LIN {X 0,Y 312.924,Z 444.508,A -85,B 0,C 180,E1 -15752.574,E2 -15752.574} C_VEL
LIN {X 0,Y 312.893,Z 444.512,A -85,B 0,C 180,E1 -15756.448,E2 -15756.448} C_VEL
LIN {X 0,Y 312.698,Z 444.535,A -85,B 0,C 180,E1 -15760.358,E2 -15760.358} C_VEL
LIN {X 0,Y 312.668,Z 444.537,A -85,B 0,C 180,E1 -15764.865,E2 -15764.865} C_VEL
LIN {X 0,Y 312.585,Z 444.545,A -85,B 0,C 180,E1 -15769.212,E2 -15769.212} C_VEL
LIN {X 0,Y 312.525,Z 444.556,A -85,B 0,C 180,E1 -15772.779,E2 -15772.779} C_VEL
LIN {X 0,Y 312.532,Z 444.552,A -85,B 0,C 180,E1 -15775.909,E2 -15775.909} C_VEL
LIN {X 0,Y 312.5,Z 444.556,A -85,B 0,C 180,E1 -15779.654,E2 -15779.654} C_VEL
LIN {X 0,Y 312.519,Z 444.553,A -85,B 0,C 180,E1 -15783.688,E2 -15783.688} C_VEL
LIN {X 0,Y 312.513,Z 444.554,A -85,B 0,C 180,E1 -15787.386,E2 -15787.386} C_VEL
LIN {X 0,Y 312.439,Z 444.567,A -85,B 0,C 180,E1 -15790.717,E2 -15790.717} C_VEL
LIN {X 0,Y 312.45,Z 444.564,A -85,B 0,C 180,E1 -15794.209,E2 -15794.209} C_VEL
LIN {X 0,Y 312.482,Z 444.558,A -85,B 0,C 180,E1 -15797.919,E2 -15797.919} C_VEL
LIN {X 0,Y 312.497,Z 444.558,A -85,B 0,C 180,E1 -15800.971,E2 -15800.971} C_VEL
LIN {X 0,Y 312.531,Z 444.554,A -85,B 0,C 180,E1 -15804.22,E2 -15804.22} C_VEL
LIN {X 0,Y 312.502,Z 444.555,A -85,B 0,C 180,E1 -15807.334,E2 -15807.334} C_VEL
LIN {X 0,Y 312.543,Z 444.55,A -85,B 0,C 180,E1 -15811.279,E2 -15811.279} C_VEL
LIN {X 0,Y 312.584,Z 444.55,A -85,B 0,C 180,E1 -15814.711,E2 -15814.711} C_VEL
LIN {X 0,Y 312.561,Z 444.546,A -85,B 0,C 180,E1 -15817.883,E2 -15817.883} C_VEL
LIN {X 0,Y 311.859,Z 444.638,A -85,B 0,C 180,E1 -15818.959,E2 -15818.959} C_VEL
LIN {X 0,Y 309.003,Z 444.996,A -85,B 0,C 180,E1 -15820.711,E2 -15820.711} C_VEL
LIN {X 0,Y 306.625,Z 445.29,A -85,B 0,C 180,E1 -15822.131,E2 -15822.131} C_VEL
LIN {X 0,Y 305.636,Z 445.412,A -85,B 0,C 180,E1 -15823.231,E2 -15823.231} C_VEL
LIN {X 0,Y 305.57,Z 445.419,A -85,B 0,C 180,E1 -15823.603,E2 -15823.603} C_VEL
LIN {X 0,Y 305.588,Z 445.421,A -85,B 0,C 180,E1 -15826.704,E2 -15826.704} C_VEL
LIN {X 0,Y 305.794,Z 445.392,A -85,B 0,C 180,E1 -15831.21,E2 -15831.21} C_VEL
LIN {X 0,Y 305.84,Z 445.385,A -85,B 0,C 180,E1 -15833.402,E2 -15833.402} C_VEL
LIN {X 0,Y 305.883,Z 445.38,A -85,B 0,C 180,E1 -15837.366,E2 -15837.366} C_VEL
LIN {X 0,Y 306.053,Z 445.359,A -85,B 0,C 180,E1 -15840,E2 -15840} C_VEL
LIN {X 0,Y 305.885,Z 445.385,A -85,B 0,C 180,E1 -15842.634,E2 -15842.634} C_VEL
LIN {X 0,Y 305.852,Z 445.388,A -85,B 0,C 180,E1 -15846.598,E2 -15846.598} C_VEL
LIN {X 0,Y 305.735,Z 445.399,A -85,B 0,C 180,E1 -15849.26,E2 -15849.26} C_VEL
LIN {X 0,Y 305.588,Z 445.417,A -85,B 0,C 180,E1 -15853.296,E2 -15853.296} C_VEL
LIN {X 0,Y 305.593,Z 445.416,A -85,B 0,C 180,E1 -15856.02,E2 -15856.02} C_VEL
LIN {X 0,Y 305.575,Z 445.418,A -85,B 0,C 180,E1 -15859.445,E2 -15859.445} C_VEL
LIN {X 0,Y 305.485,Z 445.431,A -85,B 0,C 180,E1 -15863.04,E2 -15863.04} C_VEL
LIN {X 0,Y 305.553,Z 445.422,A -85,B 0,C 180,E1 -15866.23,E2 -15866.23} C_VEL
LIN {X 0,Y 305.495,Z 445.43,A -85,B 0,C 180,E1 -15869.05,E2 -15869.05} C_VEL
LIN {X 0,Y 305.464,Z 445.432,A -85,B 0,C 180,E1 -15873.517,E2 -15873.517} C_VEL
LIN {X 0,Y 305.474,Z 445.436,A -85,B 0,C 180,E1 -15876.74,E2 -15876.74} C_VEL
LIN {X 0,Y 305.454,Z 445.437,A -85,B 0,C 180,E1 -15880.6,E2 -15880.6} C_VEL
LIN {X 0,Y 305.419,Z 445.441,A -85,B 0,C 180,E1 -15884.493,E2 -15884.493} C_VEL
LIN {X 0,Y 305.442,Z 445.435,A -85,B 0,C 180,E1 -15888.144,E2 -15888.144} C_VEL
LIN {X 0,Y 305.467,Z 445.432,A -85,B 0,C 180,E1 -15891.597,E2 -15891.597} C_VEL
LIN {X 0,Y 305.464,Z 445.437,A -85,B 0,C 180,E1 -15894.888,E2 -15894.888} C_VEL
LIN {X 0,Y 305.504,Z 445.578,A -85,B 0,C 180,E1 -15896.123,E2 -15896.123} C_VEL
LIN {X 0,Y 308.105,Z 458.028,A -85,B 0,C 180,E1 -15899.501,E2 -15899.501} C_VEL
LIN {X 0,Y 310.159,Z 467.904,A -85,B 0,C 180,E1 -15902.094,E2 -15902.094} C_VEL
LIN {X 0,Y 309.465,Z 474.625,A -85,B 0,C 180,E1 -15903.715,E2 -15903.715} C_VEL
LIN {X 0,Y 308.394,Z 483.678,A -85,B 0,C 180,E1 -15905.888,E2 -15905.888} C_VEL
LIN {X 0,Y 313.118,Z 530.091,A -85,B 0,C 180,E1 -15907.613,E2 -15907.613} C_VEL
LIN {X 0,Y 311.173,Z 594.169,A -85,B 0,C 180,E1 -15909.552,E2 -15909.552} C_VEL
LIN {X 0,Y 310.338,Z 607.85,A -85,B 0,C 180,E1 -15910.228,E2 -15910.228} C_VEL
LIN {X 0,Y 309.368,Z 620.327,A -85,B 0,C 180,E1 -15911.112,E2 -15911.112} C_VEL
LIN {X 0,Y 308.299,Z 632.472,A -85,B 0,C 180,E1 -15912.248,E2 -15912.248} C_VEL
LIN {X 0,Y 307.267,Z 643.508,A -85,B 0,C 180,E1 -15913.558,E2 -15913.558} C_VEL
LIN {X 0,Y 306.154,Z 653.974,A -85,B 0,C 180,E1 -15915.115,E2 -15915.115} C_VEL
LIN {X 0,Y 305.413,Z 662.653,A -85,B 0,C 180,E1 -15916.697,E2 -15916.697} C_VEL
LIN {X 0,Y 304.771,Z 670.189,A -85,B 0,C 180,E1 -15918.36,E2 -15918.36} C_VEL
LIN {X 0,Y 304.285,Z 677.561,A -85,B 0,C 180,E1 -15920.361,E2 -15920.361} C_VEL
LIN {X 0,Y 304.075,Z 682.515,A -85,B 0,C 180,E1 -15922.029,E2 -15922.029} C_VEL
LIN {X 0,Y 304.035,Z 687.533,A -85,B 0,C 180,E1 -15924.18,E2 -15924.18} C_VEL
LIN {X 0,Y 303.989,Z 690.733,A -85,B 0,C 180,E1 -15926.023,E2 -15926.023} C_VEL
LIN {X 0,Y 304.153,Z 692.435,A -85,B 0,C 180,E1 -15927.352,E2 -15927.352} C_VEL
LIN {X 0,Y 304.176,Z 693.668,A -85,B 0,C 180,E1 -15928.677,E2 -15928.677} C_VEL
LIN {X 0,Y 304.174,Z 694.458,A -85,B 0,C 180,E1 -15930,E2 -15930} C_VEL
LIN {X 0,Y 304.127,Z 694.76,A -85,B 0,C 180,E1 -15931.325,E2 -15931.325} C_VEL
LIN {X 0,Y 303.936,Z 694.613,A -85,B 0,C 180,E1 -15932.651,E2 -15932.651} C_VEL
LIN {X 0,Y 303.839,Z 694.053,A -85,B 0,C 180,E1 -15933.98,E2 -15933.98} C_VEL
LIN {X 0,Y 303.734,Z 692.62,A -85,B 0,C 180,E1 -15935.75,E2 -15935.75} C_VEL
LIN {X 0,Y 303.932,Z 689.733,A -85,B 0,C 180,E1 -15937.976,E2 -15937.976} C_VEL
LIN {X 0,Y 304.296,Z 686.047,A -85,B 0,C 180,E1 -15939.976,E2 -15939.976} C_VEL
LIN {X 0,Y 304.931,Z 681.285,A -85,B 0,C 180,E1 -15941.972,E2 -15941.972} C_VEL
LIN {X 0,Y 306.073,Z 675.304,A -85,B 0,C 180,E1 -15943.952,E2 -15943.952} C_VEL
LIN {X 0,Y 307.462,Z 667.925,A -85,B 0,C 180,E1 -15945.921,E2 -15945.921} C_VEL
LIN {X 0,Y 309.261,Z 658.8,A -85,B 0,C 180,E1 -15947.866,E2 -15947.866} C_VEL
LIN {X 0,Y 311.407,Z 648.631,A -85,B 0,C 180,E1 -15949.616,E2 -15949.616} C_VEL
LIN {X 0,Y 313.401,Z 638.502,A -85,B 0,C 180,E1 -15951.027,E2 -15951.027} C_VEL
LIN {X 0,Y 315.652,Z 625.934,A -85,B 0,C 180,E1 -15952.414,E2 -15952.414} C_VEL
LIN {X 0,Y 317.702,Z 613.566,A -85,B 0,C 180,E1 -15953.465,E2 -15953.465} C_VEL
LIN {X 0,Y 319.776,Z 598.2,A -85,B 0,C 180,E1 -15954.423,E2 -15954.423} C_VEL
LIN {X 0,Y 320.961,Z 584.573,A -85,B 0,C 180,E1 -15955.017,E2 -15955.017} C_VEL
LIN {X 0,Y 324.197,Z 532.422,A -85,B 0,C 180,E1 -15956.687,E2 -15956.687} C_VEL
LIN {X 0,Y 323.308,Z 519.853,A -85,B 0,C 180,E1 -15957.337,E2 -15957.337} C_VEL
LIN {X 0,Y 321.631,Z 506.064,A -85,B 0,C 180,E1 -15958.198,E2 -15958.198} C_VEL
LIN {X 0,Y 319.141,Z 492.2,A -85,B 0,C 180,E1 -15959.222,E2 -15959.222} C_VEL
LIN {X 0,Y 317.166,Z 483.192,A -85,B 0,C 180,E1 -15959.997,E2 -15959.997} C_VEL
LIN {X 0,Y 315.519,Z 479.419,A -85,B 0,C 180,E1 -15960.479,E2 -15960.479} C_VEL
LIN {X 0,Y 313.437,Z 474.649,A -85,B 0,C 180,E1 -15961.156,E2 -15961.156} C_VEL
LIN {X 0,Y 311.59,Z 466.2,A -85,B 0,C 180,E1 -15964.325,E2 -15964.325} C_VEL
LIN {X 0,Y 310.017,Z 459.968,A -85,B 0,C 180,E1 -15967.003,E2 -15967.003} C_VEL
LIN {X 0,Y 308.169,Z 453.871,A -85,B 0,C 180,E1 -15970.092,E2 -15970.092} C_VEL
LIN {X 0,Y 306.421,Z 448.344,A -85,B 0,C 180,E1 -15973.479,E2 -15973.479} C_VEL
LIN {X 0,Y 305.432,Z 445.437,A -85,B 0,C 180,E1 -15975.77,E2 -15975.77} C_VEL
LIN {X 0,Y 305.458,Z 445.433,A -85,B 0,C 180,E1 -15979.4,E2 -15979.4} C_VEL
LIN {X 0,Y 305.5,Z 445.427,A -85,B 0,C 180,E1 -15983.264,E2 -15983.264} C_VEL
LIN {X 0,Y 305.468,Z 445.435,A -85,B 0,C 180,E1 -15986.483,E2 -15986.483} C_VEL
LIN {X 0,Y 305.434,Z 445.435,A -85,B 0,C 180,E1 -15989.588,E2 -15989.588} C_VEL
LIN {X 0,Y 305.455,Z 445.437,A -85,B 0,C 180,E1 -15992.602,E2 -15992.602} C_VEL
LIN {X 0,Y 305.444,Z 445.436,A -85,B 0,C 180,E1 -15995.533,E2 -15995.533} C_VEL
LIN {X 0,Y 305.469,Z 445.479,A -85,B 0,C 180,E1 -15999.46,E2 -15999.46} C_VEL
LIN {X 0,Y 306.697,Z 449.416,A -85,B 0,C 180,E1 -16002.556,E2 -16002.556} C_VEL
LIN {X 0,Y 309.371,Z 453.214,A -85,B 0,C 180,E1 -16003.392,E2 -16003.392} C_VEL
LIN {X 0,Y 313.552,Z 459.105,A -85,B 0,C 180,E1 -16004.611,E2 -16004.611} C_VEL
LIN {X 0,Y 318.191,Z 466.055,A -85,B 0,C 180,E1 -16005.849,E2 -16005.849} C_VEL
LIN {X 0,Y 323.55,Z 475.549,A -85,B 0,C 180,E1 -16007.23,E2 -16007.23} C_VEL
LIN {X 0,Y 326.691,Z 482.075,A -85,B 0,C 180,E1 -16008.019,E2 -16008.019} C_VEL
LIN {X 0,Y 322.133,Z 551.699,A -85,B 0,C 180,E1 -16010.315,E2 -16010.315} C_VEL
LIN {X 0,Y 321.025,Z 566.069,A -85,B 0,C 180,E1 -16011.077,E2 -16011.077} C_VEL
LIN {X 0,Y 319.611,Z 579.113,A -85,B 0,C 180,E1 -16012.061,E2 -16012.061} C_VEL
LIN {X 0,Y 317.777,Z 591.737,A -85,B 0,C 180,E1 -16013.3,E2 -16013.3} C_VEL
LIN {X 0,Y 315.868,Z 603.067,A -85,B 0,C 180,E1 -16014.734,E2 -16014.734} C_VEL
LIN {X 0,Y 314.132,Z 612.119,A -85,B 0,C 180,E1 -16016.151,E2 -16016.151} C_VEL
LIN {X 0,Y 312.36,Z 620.449,A -85,B 0,C 180,E1 -16017.743,E2 -16017.743} C_VEL
LIN {X 0,Y 310.485,Z 628.539,A -85,B 0,C 180,E1 -16019.676,E2 -16019.676} C_VEL
LIN {X 0,Y 309.133,Z 634.088,A -85,B 0,C 180,E1 -16021.303,E2 -16021.303} C_VEL
LIN {X 0,Y 307.742,Z 639.484,A -85,B 0,C 180,E1 -16023.273,E2 -16023.273} C_VEL
LIN {X 0,Y 306.615,Z 643.66,A -85,B 0,C 180,E1 -16025.26,E2 -16025.26} C_VEL
LIN {X 0,Y 305.971,Z 645.843,A -85,B 0,C 180,E1 -16026.595,E2 -16026.595} C_VEL
LIN {X 0,Y 305.338,Z 647.82,A -85,B 0,C 180,E1 -16028.212,E2 -16028.212} C_VEL
LIN {X 0,Y 304.626,Z 649.586,A -85,B 0,C 180,E1 -16030.636,E2 -16030.636} C_VEL
LIN {X 0,Y 304.334,Z 649.967,A -85,B 0,C 180,E1 -16031.996,E2 -16031.996} C_VEL
LIN {X 0,Y 304.122,Z 649.714,A -85,B 0,C 180,E1 -16033.929,E2 -16033.929} C_VEL
LIN {X 0,Y 303.964,Z 648.349,A -85,B 0,C 180,E1 -16036.108,E2 -16036.108} C_VEL
LIN {X 0,Y 304.078,Z 645.291,A -85,B 0,C 180,E1 -16038.626,E2 -16038.626} C_VEL
LIN {X 0,Y 304.375,Z 640.985,A -85,B 0,C 180,E1 -16040.971,E2 -16040.971} C_VEL
LIN {X 0,Y 304.755,Z 635.706,A -85,B 0,C 180,E1 -16043.081,E2 -16043.081} C_VEL
LIN {X 0,Y 305.379,Z 628.903,A -85,B 0,C 180,E1 -16045.199,E2 -16045.199} C_VEL
LIN {X 0,Y 306.085,Z 621.556,A -85,B 0,C 180,E1 -16047.039,E2 -16047.039} C_VEL
LIN {X 0,Y 306.861,Z 613.232,A -85,B 0,C 180,E1 -16048.748,E2 -16048.748} C_VEL
LIN {X 0,Y 307.785,Z 603.69,A -85,B 0,C 180,E1 -16050.345,E2 -16050.345} C_VEL
LIN {X 0,Y 308.699,Z 593.276,A -85,B 0,C 180,E1 -16051.768,E2 -16051.768} C_VEL
LIN {X 0,Y 309.632,Z 582.052,A -85,B 0,C 180,E1 -16053.008,E2 -16053.008} C_VEL
LIN {X 0,Y 310.479,Z 569.679,A -85,B 0,C 180,E1 -16054.072,E2 -16054.072} C_VEL
LIN {X 0,Y 311.252,Z 555.875,A -85,B 0,C 180,E1 -16054.957,E2 -16054.957} C_VEL
LIN {X 0,Y 311.664,Z 543.598,A -85,B 0,C 180,E1 -16055.497,E2 -16055.497} C_VEL
LIN {X 0,Y 313.908,Z 469.49,A -85,B 0,C 180,E1 -16057.692,E2 -16057.692} C_VEL
LIN {X 0,Y 305.459,Z 445.434,A -85,B 0,C 180,E1 -16058.935,E2 -16058.935} C_VEL
LIN {X 0,Y 305.438,Z 445.439,A -85,B 0,C 180,E1 -16062.581,E2 -16062.581} C_VEL
LIN {X 0,Y 305.427,Z 445.442,A -85,B 0,C 180,E1 -16066.344,E2 -16066.344} C_VEL
LIN {X 0,Y 305.412,Z 445.44,A -85,B 0,C 180,E1 -16069.884,E2 -16069.884} C_VEL
LIN {X 0,Y 305.464,Z 445.432,A -85,B 0,C 180,E1 -16073.636,E2 -16073.636} C_VEL
LIN {X 0,Y 305.467,Z 445.437,A -85,B 0,C 180,E1 -16076.483,E2 -16076.483} C_VEL
LIN {X 0,Y 305.432,Z 445.436,A -85,B 0,C 180,E1 -16079.587,E2 -16079.587} C_VEL
LIN {X 0,Y 305.459,Z 445.436,A -85,B 0,C 180,E1 -16082.602,E2 -16082.602} C_VEL
LIN {X 0,Y 305.487,Z 445.429,A -85,B 0,C 180,E1 -16085.536,E2 -16085.536} C_VEL
LIN {X 0,Y 305.519,Z 445.426,A -85,B 0,C 180,E1 -16089.814,E2 -16089.814} C_VEL
LIN {X 0,Y 305.576,Z 445.422,A -85,B 0,C 180,E1 -16092.603,E2 -16092.603} C_VEL
LIN {X 0,Y 305.651,Z 445.409,A -85,B 0,C 180,E1 -16095.349,E2 -16095.349} C_VEL
LIN {X 0,Y 305.626,Z 445.411,A -85,B 0,C 180,E1 -16099.399,E2 -16099.399} C_VEL
LIN {X 0,Y 305.748,Z 445.398,A -85,B 0,C 180,E1 -16102.072,E2 -16102.072} C_VEL
LIN {X 0,Y 305.668,Z 445.41,A -85,B 0,C 180,E1 -16104.723,E2 -16104.723} C_VEL
LIN {X 0,Y 305.952,Z 445.374,A -85,B 0,C 180,E1 -16108.683,E2 -16108.683} C_VEL
LIN {X 0,Y 305.953,Z 445.371,A -85,B 0,C 180,E1 -16111.316,E2 -16111.316} C_VEL
LIN {X 0,Y 305.833,Z 445.39,A -85,B 0,C 180,E1 -16116.597,E2 -16116.597} C_VEL
LIN {X 0,Y 305.698,Z 445.403,A -85,B 0,C 180,E1 -16119.26,E2 -16119.26} C_VEL
LIN {X 0,Y 305.588,Z 445.417,A -85,B 0,C 180,E1 -16123.296,E2 -16123.296} C_VEL
LIN {X 0,Y 305.552,Z 445.422,A -85,B 0,C 180,E1 -16126.022,E2 -16126.022} C_VEL
LIN {X 0,Y 305.542,Z 445.422,A -85,B 0,C 180,E1 -16129.426,E2 -16129.426} C_VEL
LIN {X 0,Y 305.486,Z 445.43,A -85,B 0,C 180,E1 -16133.039,E2 -16133.039} C_VEL
LIN {X 0,Y 305.472,Z 445.433,A -85,B 0,C 180,E1 -16136.198,E2 -16136.198} C_VEL
LIN {X 0,Y 305.458,Z 445.434,A -85,B 0,C 180,E1 -16139.037,E2 -16139.037} C_VEL
LIN {X 0,Y 305.436,Z 445.436,A -85,B 0,C 180,E1 -16141.953,E2 -16141.953} C_VEL
LIN {X 0,Y 305.461,Z 445.433,A -85,B 0,C 180,E1 -16145.113,E2 -16145.113} C_VEL
LIN {X 0,Y 305.433,Z 445.441,A -85,B 0,C 180,E1 -16148.525,E2 -16148.525} C_VEL
LIN {X 0,Y 305.435,Z 445.441,A -85,B 0,C 180,E1 -16152.582,E2 -16152.582} C_VEL
LIN {X 0,Y 305.424,Z 445.44,A -85,B 0,C 180,E1 -16156.345,E2 -16156.345} C_VEL
LIN {X 0,Y 305.457,Z 445.433,A -85,B 0,C 180,E1 -16159.892,E2 -16159.892} C_VEL
LIN {X 0,Y 305.479,Z 445.43,A -85,B 0,C 180,E1 -16163.632,E2 -16163.632} C_VEL
LIN {X 0,Y 305.464,Z 445.437,A -85,B 0,C 180,E1 -16166.483,E2 -16166.483} C_VEL
LIN {X 0,Y 305.457,Z 445.432,A -85,B 0,C 180,E1 -16169.59,E2 -16169.59} C_VEL
LIN {X 0,Y 305.514,Z 445.431,A -85,B 0,C 180,E1 -16172.608,E2 -16172.608} C_VEL
LIN {X 0,Y 305.507,Z 445.427,A -85,B 0,C 180,E1 -16175.539,E2 -16175.539} C_VEL
LIN {X 0,Y 305.519,Z 445.425,A -85,B 0,C 180,E1 -16179.815,E2 -16179.815} C_VEL
LIN {X 0,Y 305.574,Z 445.424,A -85,B 0,C 180,E1 -16182.603,E2 -16182.603} C_VEL
LIN {X 0,Y 305.57,Z 445.419,A -85,B 0,C 180,E1 -16183.603,E2 -16183.603} C_VEL
LIN {X 0,Y 304.941,Z 445.502,A -85,B 0,C 180,E1 -16184.703,E2 -16184.703} C_VEL
LIN {X 0,Y 302.103,Z 445.855,A -85,B 0,C 180,E1 -16186.493,E2 -16186.493} C_VEL
LIN {X 0,Y 299.687,Z 446.154,A -85,B 0,C 180,E1 -16187.946,E2 -16187.946} C_VEL
LIN {X 0,Y 298.669,Z 446.281,A -85,B 0,C 180,E1 -16189.071,E2 -16189.071} C_VEL
LIN {X 0,Y 298.597,Z 446.287,A -85,B 0,C 180,E1 -16189.452,E2 -16189.452} C_VEL
LIN {X 0,Y 298.751,Z 446.269,A -85,B 0,C 180,E1 -16191.886,E2 -16191.886} C_VEL
LIN {X 0,Y 298.652,Z 446.286,A -85,B 0,C 180,E1 -16194.599,E2 -16194.599} C_VEL
LIN {X 0,Y 298.921,Z 446.252,A -85,B 0,C 180,E1 -16198.653,E2 -16198.653} C_VEL
LIN {X 0,Y 298.922,Z 446.247,A -85,B 0,C 180,E1 -16201.347,E2 -16201.347} C_VEL
LIN {X 0,Y 298.797,Z 446.267,A -85,B 0,C 180,E1 -16206.754,E2 -16206.754} C_VEL
LIN {X 0,Y 298.68,Z 446.277,A -85,B 0,C 180,E1 -16209.481,E2 -16209.481} C_VEL
LIN {X 0,Y 298.552,Z 446.292,A -85,B 0,C 180,E1 -16213.616,E2 -16213.616} C_VEL
LIN {X 0,Y 298.548,Z 446.296,A -85,B 0,C 180,E1 -16216.409,E2 -16216.409} C_VEL
LIN {X 0,Y 298.509,Z 446.298,A -85,B 0,C 180,E1 -16219.654,E2 -16219.654} C_VEL
LIN {X 0,Y 298.428,Z 446.308,A -85,B 0,C 180,E1 -16223.6,E2 -16223.6} C_VEL
LIN {X 0,Y 298.491,Z 446.305,A -85,B 0,C 180,E1 -16226.574,E2 -16226.574} C_VEL
LIN {X 0,Y 298.42,Z 446.309,A -85,B 0,C 180,E1 -16229.641,E2 -16229.641} C_VEL
LIN {X 0,Y 298.395,Z 446.317,A -85,B 0,C 180,E1 -16232.8,E2 -16232.8} C_VEL
LIN {X 0,Y 298.446,Z 446.311,A -85,B 0,C 180,E1 -16236.808,E2 -16236.808} C_VEL
LIN {X 0,Y 298.387,Z 446.316,A -85,B 0,C 180,E1 -16241.088,E2 -16241.088} C_VEL
LIN {X 0,Y 298.388,Z 446.316,A -85,B 0,C 180,E1 -16245.042,E2 -16245.042} C_VEL
LIN {X 0,Y 298.388,Z 446.317,A -85,B 0,C 180,E1 -16248.912,E2 -16248.912} C_VEL
LIN {X 0,Y 298.444,Z 446.309,A -85,B 0,C 180,E1 -16253.193,E2 -16253.193} C_VEL
LIN {X 0,Y 298.443,Z 446.464,A -85,B 0,C 180,E1 -16255.841,E2 -16255.841} C_VEL
LIN {X 0,Y 300.859,Z 458.098,A -85,B 0,C 180,E1 -16259.075,E2 -16259.075} C_VEL
LIN {X 0,Y 303.146,Z 468.868,A -85,B 0,C 180,E1 -16261.976,E2 -16261.976} C_VEL
LIN {X 0,Y 301.624,Z 481.991,A -85,B 0,C 180,E1 -16265.203,E2 -16265.203} C_VEL
LIN {X 0,Y 301.479,Z 483.267,A -85,B 0,C 180,E1 -16265.516,E2 -16265.516} C_VEL
LIN {X 0,Y 306.2,Z 531.288,A -85,B 0,C 180,E1 -16267.332,E2 -16267.332} C_VEL
LIN {X 0,Y 304.233,Z 593.859,A -85,B 0,C 180,E1 -16269.285,E2 -16269.285} C_VEL
LIN {X 0,Y 303.443,Z 606.759,A -85,B 0,C 180,E1 -16269.936,E2 -16269.936} C_VEL
LIN {X 0,Y 302.437,Z 619.395,A -85,B 0,C 180,E1 -16270.839,E2 -16270.839} C_VEL
LIN {X 0,Y 301.337,Z 631.609,A -85,B 0,C 180,E1 -16272,E2 -16272} C_VEL
LIN {X 0,Y 300.273,Z 642.717,A -85,B 0,C 180,E1 -16273.339,E2 -16273.339} C_VEL
LIN {X 0,Y 299.084,Z 653.754,A -85,B 0,C 180,E1 -16275.02,E2 -16275.02} C_VEL
LIN {X 0,Y 298.295,Z 662.772,A -85,B 0,C 180,E1 -16276.72,E2 -16276.72} C_VEL
LIN {X 0,Y 297.667,Z 670.193,A -85,B 0,C 180,E1 -16278.423,E2 -16278.423} C_VEL
LIN {X 0,Y 297.193,Z 677.42,A -85,B 0,C 180,E1 -16280.472,E2 -16280.472} C_VEL
LIN {X 0,Y 297.001,Z 683.144,A -85,B 0,C 180,E1 -16282.522,E2 -16282.522} C_VEL
LIN {X 0,Y 297.002,Z 687.565,A -85,B 0,C 180,E1 -16284.569,E2 -16284.569} C_VEL
LIN {X 0,Y 296.928,Z 689.844,A -85,B 0,C 180,E1 -16285.929,E2 -16285.929} C_VEL
LIN {X 0,Y 297.077,Z 691.633,A -85,B 0,C 180,E1 -16287.289,E2 -16287.289} C_VEL
LIN {X 0,Y 297.118,Z 692.919,A -85,B 0,C 180,E1 -16288.645,E2 -16288.645} C_VEL
LIN {X 0,Y 297.115,Z 693.762,A -85,B 0,C 180,E1 -16290,E2 -16290} C_VEL
LIN {X 0,Y 297.064,Z 694.158,A -85,B 0,C 180,E1 -16291.356,E2 -16291.356} C_VEL
LIN {X 0,Y 296.845,Z 694.062,A -85,B 0,C 180,E1 -16292.715,E2 -16292.715} C_VEL
LIN {X 0,Y 296.762,Z 693.548,A -85,B 0,C 180,E1 -16294.075,E2 -16294.075} C_VEL
LIN {X 0,Y 296.667,Z 692.351,A -85,B 0,C 180,E1 -16295.745,E2 -16295.745} C_VEL
LIN {X 0,Y 296.863,Z 689.43,A -85,B 0,C 180,E1 -16298.167,E2 -16298.167} C_VEL
LIN {X 0,Y 297.264,Z 685.872,A -85,B 0,C 180,E1 -16300.214,E2 -16300.214} C_VEL
LIN {X 0,Y 297.959,Z 681.219,A -85,B 0,C 180,E1 -16302.257,E2 -16302.257} C_VEL
LIN {X 0,Y 299.404,Z 674.255,A -85,B 0,C 180,E1 -16304.616,E2 -16304.616} C_VEL
LIN {X 0,Y 300.83,Z 667.312,A -85,B 0,C 180,E1 -16306.505,E2 -16306.505} C_VEL
LIN {X 0,Y 302.537,Z 659.349,A -85,B 0,C 180,E1 -16308.277,E2 -16308.277} C_VEL
LIN {X 0,Y 304.784,Z 649.381,A -85,B 0,C 180,E1 -16310.06,E2 -16310.06} C_VEL
LIN {X 0,Y 307.109,Z 638.319,A -85,B 0,C 180,E1 -16311.655,E2 -16311.655} C_VEL
LIN {X 0,Y 309.476,Z 625.993,A -85,B 0,C 180,E1 -16313.063,E2 -16313.063} C_VEL
LIN {X 0,Y 311.639,Z 613.954,A -85,B 0,C 180,E1 -16314.127,E2 -16314.127} C_VEL
LIN {X 0,Y 313.627,Z 600.459,A -85,B 0,C 180,E1 -16315.023,E2 -16315.023} C_VEL
LIN {X 0,Y 315.051,Z 586.508,A -85,B 0,C 180,E1 -16315.697,E2 -16315.697} C_VEL
LIN {X 0,Y 318.587,Z 534.067,A -85,B 0,C 180,E1 -16317.428,E2 -16317.428} C_VEL
LIN {X 0,Y 317.987,Z 522.485,A -85,B 0,C 180,E1 -16318.035,E2 -16318.035} C_VEL
LIN {X 0,Y 316.341,Z 508.34,A -85,B 0,C 180,E1 -16318.939,E2 -16318.939} C_VEL
LIN {X 0,Y 314.019,Z 494.453,A -85,B 0,C 180,E1 -16320.014,E2 -16320.014} C_VEL
LIN {X 0,Y 312.378,Z 486.751,A -85,B 0,C 180,E1 -16320.702,E2 -16320.702} C_VEL
LIN {X 0,Y 308.856,Z 479.015,A -85,B 0,C 180,E1 -16321.805,E2 -16321.805} C_VEL
LIN {X 0,Y 306.34,Z 474.117,A -85,B 0,C 180,E1 -16322.609,E2 -16322.609} C_VEL
LIN {X 0,Y 306.161,Z 473.602,A -85,B 0,C 180,E1 -16322.695,E2 -16322.695} C_VEL
LIN {X 0,Y 304.804,Z 467.402,A -85,B 0,C 180,E1 -16325.201,E2 -16325.201} C_VEL
LIN {X 0,Y 303.165,Z 461.414,A -85,B 0,C 180,E1 -16327.983,E2 -16327.983} C_VEL
LIN {X 0,Y 301.658,Z 456.346,A -85,B 0,C 180,E1 -16330.719,E2 -16330.719} C_VEL
LIN {X 0,Y 300.327,Z 452.028,A -85,B 0,C 180,E1 -16333.495,E2 -16333.495} C_VEL
LIN {X 0,Y 298.785,Z 447.863,A -85,B 0,C 180,E1 -16336.989,E2 -16336.989} C_VEL
LIN {X 0,Y 298.416,Z 446.312,A -85,B 0,C 180,E1 -16338.743,E2 -16338.743} C_VEL
LIN {X 0,Y 298.435,Z 446.312,A -85,B 0,C 180,E1 -16342.245,E2 -16342.245} C_VEL
LIN {X 0,Y 298.412,Z 446.309,A -85,B 0,C 180,E1 -16345.581,E2 -16345.581} C_VEL
LIN {X 0,Y 298.381,Z 446.317,A -85,B 0,C 180,E1 -16348.789,E2 -16348.789} C_VEL
LIN {X 0,Y 298.414,Z 446.31,A -85,B 0,C 180,E1 -16351.899,E2 -16351.899} C_VEL
LIN {X 0,Y 298.417,Z 446.315,A -85,B 0,C 180,E1 -16354.918,E2 -16354.918} C_VEL
LIN {X 0,Y 298.41,Z 446.414,A -85,B 0,C 180,E1 -16356.711,E2 -16356.711} C_VEL
LIN {X 0,Y 299.391,Z 449.481,A -85,B 0,C 180,E1 -16359.881,E2 -16359.881} C_VEL
LIN {X 0,Y 299.822,Z 450.694,A -85,B 0,C 180,E1 -16360.867,E2 -16360.867} C_VEL
LIN {X 0,Y 302.605,Z 454.462,A -85,B 0,C 180,E1 -16361.844,E2 -16361.844} C_VEL
LIN {X 0,Y 304.477,Z 457.05,A -85,B 0,C 180,E1 -16362.474,E2 -16362.474} C_VEL
LIN {X 0,Y 309.201,Z 463.406,A -85,B 0,C 180,E1 -16363.922,E2 -16363.922} C_VEL
LIN {X 0,Y 315.613,Z 473.663,A -85,B 0,C 180,E1 -16365.754,E2 -16365.754} C_VEL
LIN {X 0,Y 321.198,Z 484.416,A -85,B 0,C 180,E1 -16367.252,E2 -16367.252} C_VEL
LIN {X 0,Y 316.456,Z 552.323,A -85,B 0,C 180,E1 -16369.564,E2 -16369.564} C_VEL
LIN {X 0,Y 315.338,Z 565.985,A -85,B 0,C 180,E1 -16370.297,E2 -16370.297} C_VEL
LIN {X 0,Y 313.952,Z 578.602,A -85,B 0,C 180,E1 -16371.24,E2 -16371.24} C_VEL
LIN {X 0,Y 312.101,Z 590.826,A -85,B 0,C 180,E1 -16372.426,E2 -16372.426} C_VEL
LIN {X 0,Y 310.094,Z 602.033,A -85,B 0,C 180,E1 -16373.82,E2 -16373.82} C_VEL
LIN {X 0,Y 308.016,Z 612.21,A -85,B 0,C 180,E1 -16375.419,E2 -16375.419} C_VEL
LIN {X 0,Y 306.068,Z 620.669,A -85,B 0,C 180,E1 -16377.038,E2 -16377.038} C_VEL
LIN {X 0,Y 304.116,Z 628.855,A -85,B 0,C 180,E1 -16379.007,E2 -16379.007} C_VEL
LIN {X 0,Y 302.268,Z 635.854,A -85,B 0,C 180,E1 -16381.145,E2 -16381.145} C_VEL
LIN {X 0,Y 300.687,Z 641.419,A -85,B 0,C 180,E1 -16383.35,E2 -16383.35} C_VEL
LIN {X 0,Y 299.513,Z 645.28,A -85,B 0,C 180,E1 -16385.386,E2 -16385.386} C_VEL
LIN {X 0,Y 298.865,Z 647.225,A -85,B 0,C 180,E1 -16386.752,E2 -16386.752} C_VEL
LIN {X 0,Y 298.263,Z 648.853,A -85,B 0,C 180,E1 -16388.246,E2 -16388.246} C_VEL
LIN {X 0,Y 297.863,Z 649.81,A -85,B 0,C 180,E1 -16389.507,E2 -16389.507} C_VEL
LIN {X 0,Y 297.487,Z 650.404,A -85,B 0,C 180,E1 -16390.894,E2 -16390.894} C_VEL
LIN {X 0,Y 297.23,Z 650.572,A -85,B 0,C 180,E1 -16392.287,E2 -16392.287} C_VEL
LIN {X 0,Y 297.043,Z 650.148,A -85,B 0,C 180,E1 -16394.054,E2 -16394.054} C_VEL
LIN {X 0,Y 296.871,Z 648.371,A -85,B 0,C 180,E1 -16396.504,E2 -16396.504} C_VEL
LIN {X 0,Y 296.999,Z 645.396,A -85,B 0,C 180,E1 -16398.818,E2 -16398.818} C_VEL
LIN {X 0,Y 297.249,Z 641.809,A -85,B 0,C 180,E1 -16400.772,E2 -16400.772} C_VEL
LIN {X 0,Y 297.668,Z 636.551,A -85,B 0,C 180,E1 -16402.956,E2 -16402.956} C_VEL
LIN {X 0,Y 298.234,Z 629.886,A -85,B 0,C 180,E1 -16405.099,E2 -16405.099} C_VEL
LIN {X 0,Y 299.09,Z 621.376,A -85,B 0,C 180,E1 -16407.271,E2 -16407.271} C_VEL
LIN {X 0,Y 299.928,Z 612.441,A -85,B 0,C 180,E1 -16409.092,E2 -16409.092} C_VEL
LIN {X 0,Y 300.872,Z 603.012,A -85,B 0,C 180,E1 -16410.666,E2 -16410.666} C_VEL
LIN {X 0,Y 301.864,Z 591.901,A -85,B 0,C 180,E1 -16412.18,E2 -16412.18} C_VEL
LIN {X 0,Y 302.795,Z 579.942,A -85,B 0,C 180,E1 -16413.466,E2 -16413.466} C_VEL
LIN {X 0,Y 303.697,Z 567.093,A -85,B 0,C 180,E1 -16414.539,E2 -16414.539} C_VEL
LIN {X 0,Y 304.395,Z 553.024,A -85,B 0,C 180,E1 -16415.385,E2 -16415.385} C_VEL
LIN {X 0,Y 304.885,Z 539.253,A -85,B 0,C 180,E1 -16415.931,E2 -16415.931} C_VEL
LIN {X 0,Y 307.052,Z 470.895,A -85,B 0,C 180,E1 -16418.007,E2 -16418.007} C_VEL
LIN {X 0,Y 298.408,Z 446.311,A -85,B 0,C 180,E1 -16419.3,E2 -16419.3} C_VEL
LIN {X 0,Y 298.373,Z 446.316,A -85,B 0,C 180,E1 -16423.097,E2 -16423.097} C_VEL
LIN {X 0,Y 298.405,Z 446.312,A -85,B 0,C 180,E1 -16426.92,E2 -16426.92} C_VEL
LIN {X 0,Y 298.358,Z 446.318,A -85,B 0,C 180,E1 -16431.017,E2 -16431.017} C_VEL
LIN {X 0,Y 298.407,Z 446.312,A -85,B 0,C 180,E1 -16433.928,E2 -16433.928} C_VEL
LIN {X 0,Y 298.395,Z 446.313,A -85,B 0,C 180,E1 -16437.199,E2 -16437.199} C_VEL
LIN {X 0,Y 298.404,Z 446.315,A -85,B 0,C 180,E1 -16440.625,E2 -16440.625} C_VEL
LIN {X 0,Y 298.447,Z 446.307,A -85,B 0,C 180,E1 -16444.92,E2 -16444.92} C_VEL
LIN {X 0,Y 298.45,Z 446.306,A -85,B 0,C 180,E1 -16449.315,E2 -16449.315} C_VEL
LIN {X 0,Y 298.54,Z 446.297,A -85,B 0,C 180,E1 -16452.179,E2 -16452.179} C_VEL
LIN {X 0,Y 298.595,Z 446.289,A -85,B 0,C 180,E1 -16454.994,E2 -16454.994} C_VEL
LIN {X 0,Y 298.585,Z 446.289,A -85,B 0,C 180,E1 -16459.146,E2 -16459.146} C_VEL
LIN {X 0,Y 298.699,Z 446.275,A -85,B 0,C 180,E1 -16461.884,E2 -16461.884} C_VEL
LIN {X 0,Y 298.637,Z 446.287,A -85,B 0,C 180,E1 -16464.598,E2 -16464.598} C_VEL
LIN {X 0,Y 298.919,Z 446.25,A -85,B 0,C 180,E1 -16468.652,E2 -16468.652} C_VEL
LIN {X 0,Y 298.919,Z 446.247,A -85,B 0,C 180,E1 -16471.347,E2 -16471.347} C_VEL
LIN {X 0,Y 298.777,Z 446.267,A -85,B 0,C 180,E1 -16476.754,E2 -16476.754} C_VEL
LIN {X 0,Y 298.631,Z 446.283,A -85,B 0,C 180,E1 -16479.482,E2 -16479.482} C_VEL
LIN {X 0,Y 298.546,Z 446.294,A -85,B 0,C 180,E1 -16483.615,E2 -16483.615} C_VEL
LIN {X 0,Y 298.487,Z 446.305,A -85,B 0,C 180,E1 -16486.412,E2 -16486.412} C_VEL
LIN {X 0,Y 298.483,Z 446.302,A -85,B 0,C 180,E1 -16489.639,E2 -16489.639} C_VEL
LIN {X 0,Y 298.423,Z 446.309,A -85,B 0,C 180,E1 -16493.6,E2 -16493.6} C_VEL
LIN {X 0,Y 298.412,Z 446.315,A -85,B 0,C 180,E1 -16496.581,E2 -16496.581} C_VEL
LIN {X 0,Y 298.397,Z 446.312,A -85,B 0,C 180,E1 -16499.643,E2 -16499.643} C_VEL
LIN {X 0,Y 298.392,Z 446.315,A -85,B 0,C 180,E1 -16502.8,E2 -16502.8} C_VEL
LIN {X 0,Y 298.441,Z 446.31,A -85,B 0,C 180,E1 -16506.806,E2 -16506.806} C_VEL
LIN {X 0,Y 298.347,Z 446.319,A -85,B 0,C 180,E1 -16511.079,E2 -16511.079} C_VEL
LIN {X 0,Y 298.398,Z 446.313,A -85,B 0,C 180,E1 -16513.103,E2 -16513.103} C_VEL
LIN {X 0,Y 298.402,Z 446.314,A -85,B 0,C 180,E1 -16516.92,E2 -16516.92} C_VEL
LIN {X 0,Y 298.397,Z 446.313,A -85,B 0,C 180,E1 -16521.007,E2 -16521.007} C_VEL
LIN {X 0,Y 298.417,Z 446.31,A -85,B 0,C 180,E1 -16523.93,E2 -16523.93} C_VEL
LIN {X 0,Y 298.392,Z 446.314,A -85,B 0,C 180,E1 -16527.984,E2 -16527.984} C_VEL
LIN {X 0,Y 298.456,Z 446.305,A -85,B 0,C 180,E1 -16531.904,E2 -16531.904} C_VEL
LIN {X 0,Y 298.482,Z 446.304,A -85,B 0,C 180,E1 -16534.924,E2 -16534.924} C_VEL
LIN {X 0,Y 298.45,Z 446.306,A -85,B 0,C 180,E1 -16539.315,E2 -16539.315} C_VEL
LIN {X 0,Y 298.537,Z 446.297,A -85,B 0,C 180,E1 -16542.179,E2 -16542.179} C_VEL
LIN {X 0,Y 298.593,Z 446.29,A -85,B 0,C 180,E1 -16544.995,E2 -16544.995} C_VEL
LIN {X 0,Y 298.597,Z 446.287,A -85,B 0,C 180,E1 -16549.452,E2 -16549.452} C_VEL
LIN {X 0,Y 297.962,Z 446.371,A -85,B 0,C 180,E1 -16550.58,E2 -16550.58} C_VEL
LIN {X 0,Y 295.129,Z 446.723,A -85,B 0,C 180,E1 -16552.416,E2 -16552.416} C_VEL
LIN {X 0,Y 292.699,Z 447.023,A -85,B 0,C 180,E1 -16553.906,E2 -16553.906} C_VEL
LIN {X 0,Y 291.644,Z 447.155,A -85,B 0,C 180,E1 -16555.06,E2 -16555.06} C_VEL
LIN {X 0,Y 291.552,Z 447.164,A -85,B 0,C 180,E1 -16555.452,E2 -16555.452} C_VEL
LIN {X 0,Y 291.888,Z 447.128,A -85,B 0,C 180,E1 -16558.62,E2 -16558.62} C_VEL
LIN {X 0,Y 291.888,Z 447.124,A -85,B 0,C 180,E1 -16561.38,E2 -16561.38} C_VEL
LIN {X 0,Y 291.746,Z 447.144,A -85,B 0,C 180,E1 -16566.918,E2 -16566.918} C_VEL
LIN {X 0,Y 291.629,Z 447.156,A -85,B 0,C 180,E1 -16569.712,E2 -16569.712} C_VEL
LIN {X 0,Y 291.521,Z 447.168,A -85,B 0,C 180,E1 -16573.95,E2 -16573.95} C_VEL
LIN {X 0,Y 291.487,Z 447.177,A -85,B 0,C 180,E1 -16576.818,E2 -16576.818} C_VEL
LIN {X 0,Y 291.45,Z 447.178,A -85,B 0,C 180,E1 -16579.875,E2 -16579.875} C_VEL
LIN {X 0,Y 291.382,Z 447.187,A -85,B 0,C 180,E1 -16584.207,E2 -16584.207} C_VEL
LIN {X 0,Y 291.425,Z 447.182,A -85,B 0,C 180,E1 -16587.271,E2 -16587.271} C_VEL
LIN {X 0,Y 291.337,Z 447.194,A -85,B 0,C 180,E1 -16590.437,E2 -16590.437} C_VEL
LIN {X 0,Y 291.344,Z 447.191,A -85,B 0,C 180,E1 -16593.699,E2 -16593.699} C_VEL
LIN {X 0,Y 291.375,Z 447.188,A -85,B 0,C 180,E1 -16597.254,E2 -16597.254} C_VEL
LIN {X 0,Y 291.333,Z 447.196,A -85,B 0,C 180,E1 -16600.643,E2 -16600.643} C_VEL
LIN {X 0,Y 291.314,Z 447.197,A -85,B 0,C 180,E1 -16604.398,E2 -16604.398} C_VEL
LIN {X 0,Y 291.327,Z 447.195,A -85,B 0,C 180,E1 -16608.404,E2 -16608.404} C_VEL
LIN {X 0,Y 291.348,Z 447.192,A -85,B 0,C 180,E1 -16611.158,E2 -16611.158} C_VEL
LIN {X 0,Y 291.361,Z 447.194,A -85,B 0,C 180,E1 -16614.627,E2 -16614.627} C_VEL
LIN {X 0,Y 291.39,Z 447.347,A -85,B 0,C 180,E1 -16615.551,E2 -16615.551} C_VEL
LIN {X 0,Y 293.805,Z 458.959,A -85,B 0,C 180,E1 -16618.861,E2 -16618.861} C_VEL
LIN {X 0,Y 295.977,Z 469.063,A -85,B 0,C 180,E1 -16621.647,E2 -16621.647} C_VEL
LIN {X 0,Y 295.964,Z 472.034,A -85,B 0,C 180,E1 -16622.416,E2 -16622.416} C_VEL
LIN {X 0,Y 294.56,Z 482.693,A -85,B 0,C 180,E1 -16625.101,E2 -16625.101} C_VEL
LIN {X 0,Y 299.303,Z 531.58,A -85,B 0,C 180,E1 -16627.014,E2 -16627.014} C_VEL
LIN {X 0,Y 297.292,Z 593.168,A -85,B 0,C 180,E1 -16629.005,E2 -16629.005} C_VEL
LIN {X 0,Y 296.453,Z 606.738,A -85,B 0,C 180,E1 -16629.714,E2 -16629.714} C_VEL
LIN {X 0,Y 295.505,Z 618.206,A -85,B 0,C 180,E1 -16630.552,E2 -16630.552} C_VEL
LIN {X 0,Y 294.373,Z 630.51,A -85,B 0,C 180,E1 -16631.739,E2 -16631.739} C_VEL
LIN {X 0,Y 293.286,Z 641.704,A -85,B 0,C 180,E1 -16633.11,E2 -16633.11} C_VEL
LIN {X 0,Y 292.195,Z 651.844,A -85,B 0,C 180,E1 -16634.659,E2 -16634.659} C_VEL
LIN {X 0,Y 291.347,Z 661.082,A -85,B 0,C 180,E1 -16636.397,E2 -16636.397} C_VEL
LIN {X 0,Y 290.56,Z 670.08,A -85,B 0,C 180,E1 -16638.49,E2 -16638.49} C_VEL
LIN {X 0,Y 290.122,Z 677.211,A -85,B 0,C 180,E1 -16640.59,E2 -16640.59} C_VEL
LIN {X 0,Y 289.929,Z 683.7,A -85,B 0,C 180,E1 -16643.039,E2 -16643.039} C_VEL
LIN {X 0,Y 289.906,Z 687.842,A -85,B 0,C 180,E1 -16645.133,E2 -16645.133} C_VEL
LIN {X 0,Y 290.004,Z 690.814,A -85,B 0,C 180,E1 -16647.222,E2 -16647.222} C_VEL
LIN {X 0,Y 290.061,Z 692.17,A -85,B 0,C 180,E1 -16648.612,E2 -16648.612} C_VEL
LIN {X 0,Y 290.056,Z 693.064,A -85,B 0,C 180,E1 -16650.001,E2 -16650.001} C_VEL
LIN {X 0,Y 290,Z 693.521,A -85,B 0,C 180,E1 -16651.389,E2 -16651.389} C_VEL
LIN {X 0,Y 289.755,Z 693.51,A -85,B 0,C 180,E1 -16652.781,E2 -16652.781} C_VEL
LIN {X 0,Y 289.684,Z 693.048,A -85,B 0,C 180,E1 -16654.174,E2 -16654.174} C_VEL
LIN {X 0,Y 289.595,Z 692.051,A -85,B 0,C 180,E1 -16655.728,E2 -16655.728} C_VEL
LIN {X 0,Y 289.816,Z 689.148,A -85,B 0,C 180,E1 -16658.367,E2 -16658.367} C_VEL
LIN {X 0,Y 290.246,Z 685.697,A -85,B 0,C 180,E1 -16660.464,E2 -16660.464} C_VEL
LIN {X 0,Y 291.003,Z 681.173,A -85,B 0,C 180,E1 -16662.555,E2 -16662.555} C_VEL
LIN {X 0,Y 292.516,Z 674.404,A -85,B 0,C 180,E1 -16664.969,E2 -16664.969} C_VEL
LIN {X 0,Y 294.292,Z 666.419,A -85,B 0,C 180,E1 -16667.206,E2 -16667.206} C_VEL
LIN {X 0,Y 296.217,Z 658.212,A -85,B 0,C 180,E1 -16669.041,E2 -16669.041} C_VEL
LIN {X 0,Y 298.872,Z 647.223,A -85,B 0,C 180,E1 -16671.015,E2 -16671.015} C_VEL
LIN {X 0,Y 301.4,Z 635.882,A -85,B 0,C 180,E1 -16672.628,E2 -16672.628} C_VEL
LIN {X 0,Y 303.66,Z 624.705,A -85,B 0,C 180,E1 -16673.893,E2 -16673.893} C_VEL
LIN {X 0,Y 305.928,Z 612.52,A -85,B 0,C 180,E1 -16674.969,E2 -16674.969} C_VEL
LIN {X 0,Y 308.202,Z 597.515,A -85,B 0,C 180,E1 -16675.947,E2 -16675.947} C_VEL
LIN {X 0,Y 309.535,Z 584.73,A -85,B 0,C 180,E1 -16676.552,E2 -16676.552} C_VEL
LIN {X 0,Y 313.153,Z 534.03,A -85,B 0,C 180,E1 -16678.273,E2 -16678.273} C_VEL
LIN {X 0,Y 312.416,Z 521.681,A -85,B 0,C 180,E1 -16678.971,E2 -16678.971} C_VEL
LIN {X 0,Y 310.814,Z 508.009,A -85,B 0,C 180,E1 -16679.926,E2 -16679.926} C_VEL
LIN {X 0,Y 308.667,Z 495.05,A -85,B 0,C 180,E1 -16680.982,E2 -16680.982} C_VEL
LIN {X 0,Y 307.551,Z 489.988,A -85,B 0,C 180,E1 -16681.482,E2 -16681.482} C_VEL
LIN {X 0,Y 304.248,Z 482.958,A -85,B 0,C 180,E1 -16682.578,E2 -16682.578} C_VEL
LIN {X 0,Y 301.571,Z 477.69,A -85,B 0,C 180,E1 -16683.501,E2 -16683.501} C_VEL
LIN {X 0,Y 298.806,Z 472.154,A -85,B 0,C 180,E1 -16684.592,E2 -16684.592} C_VEL
LIN {X 0,Y 297.495,Z 466.704,A -85,B 0,C 180,E1 -16687.073,E2 -16687.073} C_VEL
LIN {X 0,Y 295.644,Z 460.356,A -85,B 0,C 180,E1 -16690.474,E2 -16690.474} C_VEL
LIN {X 0,Y 294.07,Z 455.244,A -85,B 0,C 180,E1 -16693.875,E2 -16693.875} C_VEL
LIN {X 0,Y 292.507,Z 450.486,A -85,B 0,C 180,E1 -16698.145,E2 -16698.145} C_VEL
LIN {X 0,Y 291.442,Z 447.18,A -85,B 0,C 180,E1 -16703.141,E2 -16703.141} C_VEL
LIN {X 0,Y 291.347,Z 447.192,A -85,B 0,C 180,E1 -16706.302,E2 -16706.302} C_VEL
LIN {X 0,Y 291.368,Z 447.188,A -85,B 0,C 180,E1 -16710.268,E2 -16710.268} C_VEL
LIN {X 0,Y 291.381,Z 447.206,A -85,B 0,C 180,E1 -16711.944,E2 -16711.944} C_VEL
LIN {X 0,Y 292.108,Z 449.624,A -85,B 0,C 180,E1 -16716.103,E2 -16716.103} C_VEL
LIN {X 0,Y 293.002,Z 452.156,A -85,B 0,C 180,E1 -16718.912,E2 -16718.912} C_VEL
LIN {X 0,Y 296.079,Z 456.135,A -85,B 0,C 180,E1 -16720.159,E2 -16720.159} C_VEL
LIN {X 0,Y 297.457,Z 457.853,A -85,B 0,C 180,E1 -16720.684,E2 -16720.684} C_VEL
LIN {X 0,Y 300.754,Z 462.181,A -85,B 0,C 180,E1 -16721.858,E2 -16721.858} C_VEL
LIN {X 0,Y 305.941,Z 469.64,A -85,B 0,C 180,E1 -16723.564,E2 -16723.564} C_VEL
LIN {X 0,Y 311.404,Z 478.539,A -85,B 0,C 180,E1 -16725.207,E2 -16725.207} C_VEL
LIN {X 0,Y 315.871,Z 487.382,A -85,B 0,C 180,E1 -16726.481,E2 -16726.481} C_VEL
LIN {X 0,Y 310.934,Z 552.95,A -85,B 0,C 180,E1 -16728.758,E2 -16728.758} C_VEL
LIN {X 0,Y 309.67,Z 567.101,A -85,B 0,C 180,E1 -16729.539,E2 -16729.539} C_VEL
LIN {X 0,Y 308.199,Z 579.335,A -85,B 0,C 180,E1 -16730.484,E2 -16730.484} C_VEL
LIN {X 0,Y 306.165,Z 591.905,A -85,B 0,C 180,E1 -16731.739,E2 -16731.739} C_VEL
LIN {X 0,Y 304.244,Z 602.185,A -85,B 0,C 180,E1 -16733.034,E2 -16733.034} C_VEL
LIN {X 0,Y 301.999,Z 612.487,A -85,B 0,C 180,E1 -16734.659,E2 -16734.659} C_VEL
LIN {X 0,Y 299.913,Z 620.951,A -85,B 0,C 180,E1 -16736.305,E2 -16736.305} C_VEL
LIN {X 0,Y 297.777,Z 629.183,A -85,B 0,C 180,E1 -16738.309,E2 -16738.309} C_VEL
LIN {X 0,Y 295.879,Z 635.853,A -85,B 0,C 180,E1 -16740.349,E2 -16740.349} C_VEL
LIN {X 0,Y 294.064,Z 641.879,A -85,B 0,C 180,E1 -16742.74,E2 -16742.74} C_VEL
LIN {X 0,Y 292.772,Z 645.769,A -85,B 0,C 180,E1 -16744.819,E2 -16744.819} C_VEL
LIN {X 0,Y 291.76,Z 648.565,A -85,B 0,C 180,E1 -16746.918,E2 -16746.918} C_VEL
LIN {X 0,Y 291.174,Z 649.861,A -85,B 0,C 180,E1 -16748.327,E2 -16748.327} C_VEL
LIN {X 0,Y 290.732,Z 650.717,A -85,B 0,C 180,E1 -16749.742,E2 -16749.742} C_VEL
LIN {X 0,Y 290.373,Z 651.156,A -85,B 0,C 180,E1 -16751.164,E2 -16751.164} C_VEL
LIN {X 0,Y 290.109,Z 651.127,A -85,B 0,C 180,E1 -16752.593,E2 -16752.593} C_VEL
LIN {X 0,Y 289.948,Z 650.567,A -85,B 0,C 180,E1 -16754.172,E2 -16754.172} C_VEL
LIN {X 0,Y 289.809,Z 649.722,A -85,B 0,C 180,E1 -16755.471,E2 -16755.471} C_VEL
LIN {X 0,Y 289.782,Z 648.32,A -85,B 0,C 180,E1 -16756.92,E2 -16756.92} C_VEL
LIN {X 0,Y 289.93,Z 645.429,A -85,B 0,C 180,E1 -16759.024,E2 -16759.024} C_VEL
LIN {X 0,Y 290.241,Z 641.071,A -85,B 0,C 180,E1 -16761.298,E2 -16761.298} C_VEL
LIN {X 0,Y 290.712,Z 635.187,A -85,B 0,C 180,E1 -16763.612,E2 -16763.612} C_VEL
LIN {X 0,Y 291.389,Z 628.299,A -85,B 0,C 180,E1 -16765.731,E2 -16765.731} C_VEL
LIN {X 0,Y 292.27,Z 619.12,A -85,B 0,C 180,E1 -16767.963,E2 -16767.963} C_VEL
LIN {X 0,Y 293.231,Z 609.579,A -85,B 0,C 180,E1 -16769.823,E2 -16769.823} C_VEL
LIN {X 0,Y 294.201,Z 598.716,A -85,B 0,C 180,E1 -16771.528,E2 -16771.528} C_VEL
LIN {X 0,Y 295.272,Z 587.094,A -85,B 0,C 180,E1 -16772.988,E2 -16772.988} C_VEL
LIN {X 0,Y 296.318,Z 573.957,A -85,B 0,C 180,E1 -16774.269,E2 -16774.269} C_VEL
LIN {X 0,Y 297.112,Z 561.174,A -85,B 0,C 180,E1 -16775.21,E2 -16775.21} C_VEL
LIN {X 0,Y 297.723,Z 546.639,A -85,B 0,C 180,E1 -16775.958,E2 -16775.958} C_VEL
LIN {X 0,Y 300.124,Z 472.17,A -85,B 0,C 180,E1 -16778.326,E2 -16778.326} C_VEL
LIN {X 0,Y 291.354,Z 447.191,A -85,B 0,C 180,E1 -16779.685,E2 -16779.685} C_VEL
LIN {X 0,Y 291.292,Z 447.198,A -85,B 0,C 180,E1 -16783.629,E2 -16783.629} C_VEL
LIN {X 0,Y 291.314,Z 447.194,A -85,B 0,C 180,E1 -16787.506,E2 -16787.506} C_VEL
LIN {X 0,Y 291.311,Z 447.195,A -85,B 0,C 180,E1 -16791.151,E2 -16791.151} C_VEL
LIN {X 0,Y 291.357,Z 447.192,A -85,B 0,C 180,E1 -16794.625,E2 -16794.625} C_VEL
LIN {X 0,Y 291.368,Z 447.189,A -85,B 0,C 180,E1 -16797.95,E2 -16797.95} C_VEL
LIN {X 0,Y 291.346,Z 447.191,A -85,B 0,C 180,E1 -16801.154,E2 -16801.154} C_VEL
LIN {X 0,Y 291.364,Z 447.191,A -85,B 0,C 180,E1 -16804.266,E2 -16804.266} C_VEL
LIN {X 0,Y 291.379,Z 447.187,A -85,B 0,C 180,E1 -16807.299,E2 -16807.299} C_VEL
LIN {X 0,Y 291.46,Z 447.18,A -85,B 0,C 180,E1 -16810.27,E2 -16810.27} C_VEL
LIN {X 0,Y 291.557,Z 447.168,A -85,B 0,C 180,E1 -16814.623,E2 -16814.623} C_VEL
LIN {X 0,Y 291.531,Z 447.169,A -85,B 0,C 180,E1 -16818.88,E2 -16818.88} C_VEL
LIN {X 0,Y 291.653,Z 447.152,A -85,B 0,C 180,E1 -16821.686,E2 -16821.686} C_VEL
LIN {X 0,Y 291.606,Z 447.164,A -85,B 0,C 180,E1 -16824.467,E2 -16824.467} C_VEL
LIN {X 0,Y 291.885,Z 447.127,A -85,B 0,C 180,E1 -16828.62,E2 -16828.62} C_VEL
LIN {X 0,Y 291.886,Z 447.123,A -85,B 0,C 180,E1 -16831.379,E2 -16831.379} C_VEL
LIN {X 0,Y 291.724,Z 447.144,A -85,B 0,C 180,E1 -16836.918,E2 -16836.918} C_VEL
LIN {X 0,Y 291.573,Z 447.162,A -85,B 0,C 180,E1 -16839.713,E2 -16839.713} C_VEL
LIN {X 0,Y 291.516,Z 447.17,A -85,B 0,C 180,E1 -16843.95,E2 -16843.95} C_VEL
LIN {X 0,Y 291.44,Z 447.181,A -85,B 0,C 180,E1 -16848.269,E2 -16848.269} C_VEL
LIN {X 0,Y 291.359,Z 447.19,A -85,B 0,C 180,E1 -16851.212,E2 -16851.212} C_VEL
LIN {X 0,Y 291.365,Z 447.19,A -85,B 0,C 180,E1 -16854.208,E2 -16854.208} C_VEL
LIN {X 0,Y 291.358,Z 447.189,A -85,B 0,C 180,E1 -16857.278,E2 -16857.278} C_VEL
LIN {X 0,Y 291.32,Z 447.198,A -85,B 0,C 180,E1 -16860.438,E2 -16860.438} C_VEL
LIN {X 0,Y 291.343,Z 447.19,A -85,B 0,C 180,E1 -16863.698,E2 -16863.698} C_VEL
LIN {X 0,Y 291.367,Z 447.189,A -85,B 0,C 180,E1 -16867.252,E2 -16867.252} C_VEL
LIN {X 0,Y 291.299,Z 447.201,A -85,B 0,C 180,E1 -16870.648,E2 -16870.648} C_VEL
LIN {X 0,Y 291.289,Z 447.201,A -85,B 0,C 180,E1 -16874.402,E2 -16874.402} C_VEL
LIN {X 0,Y 291.325,Z 447.197,A -85,B 0,C 180,E1 -16878.404,E2 -16878.404} C_VEL
LIN {X 0,Y 291.346,Z 447.191,A -85,B 0,C 180,E1 -16881.157,E2 -16881.157} C_VEL
LIN {X 0,Y 291.36,Z 447.194,A -85,B 0,C 180,E1 -16884.626,E2 -16884.626} C_VEL
LIN {X 0,Y 291.369,Z 447.188,A -85,B 0,C 180,E1 -16887.95,E2 -16887.95} C_VEL
LIN {X 0,Y 291.376,Z 447.188,A -85,B 0,C 180,E1 -16891.158,E2 -16891.158} C_VEL
LIN {X 0,Y 291.411,Z 447.185,A -85,B 0,C 180,E1 -16894.271,E2 -16894.271} C_VEL
LIN {X 0,Y 291.381,Z 447.186,A -85,B 0,C 180,E1 -16897.3,E2 -16897.3} C_VEL
LIN {X 0,Y 291.457,Z 447.178,A -85,B 0,C 180,E1 -16900.27,E2 -16900.27} C_VEL
LIN {X 0,Y 291.554,Z 447.17,A -85,B 0,C 180,E1 -16904.624,E2 -16904.624} C_VEL
LIN {X 0,Y 291.536,Z 447.17,A -85,B 0,C 180,E1 -16908.881,E2 -16908.881} C_VEL
LIN {X 0,Y 291.703,Z 447.146,A -85,B 0,C 180,E1 -16911.688,E2 -16911.688} C_VEL
LIN {X 0,Y 291.623,Z 447.16,A -85,B 0,C 180,E1 -16914.468,E2 -16914.468} C_VEL
LIN {X 0,Y 291.552,Z 447.164,A -85,B 0,C 180,E1 -16915.452,E2 -16915.452} C_VEL
LIN {X 0,Y 290.923,Z 447.247,A -85,B 0,C 180,E1 -16916.607,E2 -16916.607} C_VEL
LIN {X 0,Y 288.275,Z 447.577,A -85,B 0,C 180,E1 -16918.495,E2 -16918.495} C_VEL
LIN {X 0,Y 285.195,Z 447.961,A -85,B 0,C 180,E1 -16920.809,E2 -16920.809} C_VEL
LIN {X 0,Y 284.829,Z 448.002,A -85,B 0,C 180,E1 -16921.607,E2 -16921.607} C_VEL
LIN {X 0,Y 284.698,Z 448.02,A -85,B 0,C 180,E1 -16927.09,E2 -16927.09} C_VEL
LIN {X 0,Y 284.566,Z 448.036,A -85,B 0,C 180,E1 -16929.955,E2 -16929.955} C_VEL
LIN {X 0,Y 284.481,Z 448.047,A -85,B 0,C 180,E1 -16934.303,E2 -16934.303} C_VEL
LIN {X 0,Y 284.425,Z 448.054,A -85,B 0,C 180,E1 -16937.249,E2 -16937.249} C_VEL
LIN {X 0,Y 284.377,Z 448.06,A -85,B 0,C 180,E1 -16940.243,E2 -16940.243} C_VEL
LIN {X 0,Y 284.339,Z 448.067,A -85,B 0,C 180,E1 -16944.847,E2 -16944.847} C_VEL
LIN {X 0,Y 284.334,Z 448.065,A -85,B 0,C 180,E1 -16948.01,E2 -16948.01} C_VEL
LIN {X 0,Y 284.295,Z 448.069,A -85,B 0,C 180,E1 -16951.275,E2 -16951.275} C_VEL
LIN {X 0,Y 284.34,Z 448.064,A -85,B 0,C 180,E1 -16955.348,E2 -16955.348} C_VEL
LIN {X 0,Y 284.312,Z 448.068,A -85,B 0,C 180,E1 -16958.169,E2 -16958.169} C_VEL
LIN {X 0,Y 284.269,Z 448.073,A -85,B 0,C 180,E1 -16962.125,E2 -16962.125} C_VEL
LIN {X 0,Y 284.268,Z 448.073,A -85,B 0,C 180,E1 -16966.192,E2 -16966.192} C_VEL
LIN {X 0,Y 284.306,Z 448.067,A -85,B 0,C 180,E1 -16970.024,E2 -16970.024} C_VEL
LIN {X 0,Y 284.331,Z 448.066,A -85,B 0,C 180,E1 -16973.614,E2 -16973.614} C_VEL
LIN {X 0,Y 284.364,Z 448.251,A -85,B 0,C 180,E1 -16975.271,E2 -16975.271} C_VEL
LIN {X 0,Y 286.991,Z 461.008,A -85,B 0,C 180,E1 -16978.993,E2 -16978.993} C_VEL
LIN {X 0,Y 289.027,Z 470.681,A -85,B 0,C 180,E1 -16981.713,E2 -16981.713} C_VEL
LIN {X 0,Y 288.074,Z 479.32,A -85,B 0,C 180,E1 -16983.952,E2 -16983.952} C_VEL
LIN {X 0,Y 287.661,Z 482.325,A -85,B 0,C 180,E1 -16984.726,E2 -16984.726} C_VEL
LIN {X 0,Y 292.065,Z 527.706,A -85,B 0,C 180,E1 -16986.55,E2 -16986.55} C_VEL
LIN {X 0,Y 292.338,Z 533.52,A -85,B 0,C 180,E1 -16986.762,E2 -16986.762} C_VEL
LIN {X 0,Y 290.339,Z 592.146,A -85,B 0,C 180,E1 -16988.71,E2 -16988.71} C_VEL
LIN {X 0,Y 289.568,Z 605.151,A -85,B 0,C 180,E1 -16989.395,E2 -16989.395} C_VEL
LIN {X 0,Y 288.56,Z 616.856,A -85,B 0,C 180,E1 -16990.25,E2 -16990.25} C_VEL
LIN {X 0,Y 287.412,Z 629.36,A -85,B 0,C 180,E1 -16991.465,E2 -16991.465} C_VEL
LIN {X 0,Y 286.291,Z 640.657,A -85,B 0,C 180,E1 -16992.868,E2 -16992.868} C_VEL
LIN {X 0,Y 285.209,Z 650.928,A -85,B 0,C 180,E1 -16994.457,E2 -16994.457} C_VEL
LIN {X 0,Y 284.23,Z 661.061,A -85,B 0,C 180,E1 -16996.415,E2 -16996.415} C_VEL
LIN {X 0,Y 283.58,Z 668.596,A -85,B 0,C 180,E1 -16998.203,E2 -16998.203} C_VEL
LIN {X 0,Y 283.071,Z 675.953,A -85,B 0,C 180,E1 -17000.353,E2 -17000.353} C_VEL
LIN {X 0,Y 282.875,Z 680.898,A -85,B 0,C 180,E1 -17002.147,E2 -17002.147} C_VEL
LIN {X 0,Y 282.893,Z 685.605,A -85,B 0,C 180,E1 -17004.297,E2 -17004.297} C_VEL
LIN {X 0,Y 282.811,Z 688.009,A -85,B 0,C 180,E1 -17005.725,E2 -17005.725} C_VEL
LIN {X 0,Y 282.934,Z 689.949,A -85,B 0,C 180,E1 -17007.153,E2 -17007.153} C_VEL
LIN {X 0,Y 283.005,Z 691.407,A -85,B 0,C 180,E1 -17008.578,E2 -17008.578} C_VEL
LIN {X 0,Y 283,Z 692.352,A -85,B 0,C 180,E1 -17010.001,E2 -17010.001} C_VEL
LIN {X 0,Y 282.936,Z 692.86,A -85,B 0,C 180,E1 -17011.424,E2 -17011.424} C_VEL
LIN {X 0,Y 282.668,Z 692.922,A -85,B 0,C 180,E1 -17012.851,E2 -17012.851} C_VEL
LIN {X 0,Y 282.586,Z 692.552,A -85,B 0,C 180,E1 -17014.279,E2 -17014.279} C_VEL
LIN {X 0,Y 282.524,Z 691.729,A -85,B 0,C 180,E1 -17015.711,E2 -17015.711} C_VEL
LIN {X 0,Y 282.547,Z 690.492,A -85,B 0,C 180,E1 -17017.145,E2 -17017.145} C_VEL
LIN {X 0,Y 282.862,Z 687.832,A -85,B 0,C 180,E1 -17019.294,E2 -17019.294} C_VEL
LIN {X 0,Y 283.431,Z 684.172,A -85,B 0,C 180,E1 -17021.442,E2 -17021.442} C_VEL
LIN {X 0,Y 284.503,Z 679.423,A -85,B 0,C 180,E1 -17023.573,E2 -17023.573} C_VEL
LIN {X 0,Y 286.106,Z 672.368,A -85,B 0,C 180,E1 -17026.043,E2 -17026.043} C_VEL
LIN {X 0,Y 288.016,Z 664.792,A -85,B 0,C 180,E1 -17028.13,E2 -17028.13} C_VEL
LIN {X 0,Y 290.418,Z 655.548,A -85,B 0,C 180,E1 -17030.173,E2 -17030.173} C_VEL
LIN {X 0,Y 293.036,Z 645.149,A -85,B 0,C 180,E1 -17032.009,E2 -17032.009} C_VEL
LIN {X 0,Y 295.77,Z 633.442,A -85,B 0,C 180,E1 -17033.64,E2 -17033.64} C_VEL
LIN {X 0,Y 298.265,Z 622.025,A -85,B 0,C 180,E1 -17034.91,E2 -17034.91} C_VEL
LIN {X 0,Y 300.757,Z 609.304,A -85,B 0,C 180,E1 -17035.986,E2 -17035.986} C_VEL
LIN {X 0,Y 302.746,Z 596.384,A -85,B 0,C 180,E1 -17036.823,E2 -17036.823} C_VEL
LIN {X 0,Y 304.154,Z 583.37,A -85,B 0,C 180,E1 -17037.432,E2 -17037.432} C_VEL
LIN {X 0,Y 307.817,Z 535.046,A -85,B 0,C 180,E1 -17039.124,E2 -17039.124} C_VEL
LIN {X 0,Y 307.154,Z 522.209,A -85,B 0,C 180,E1 -17039.884,E2 -17039.884} C_VEL
LIN {X 0,Y 305.182,Z 505.597,A -85,B 0,C 180,E1 -17041.122,E2 -17041.122} C_VEL
LIN {X 0,Y 303.129,Z 494.061,A -85,B 0,C 180,E1 -17042.192,E2 -17042.192} C_VEL
LIN {X 0,Y 300.258,Z 487.884,A -85,B 0,C 180,E1 -17043.198,E2 -17043.198} C_VEL
LIN {X 0,Y 297.686,Z 482.611,A -85,B 0,C 180,E1 -17044.162,E2 -17044.162} C_VEL
LIN {X 0,Y 294.599,Z 476.754,A -85,B 0,C 180,E1 -17045.36,E2 -17045.36} C_VEL
LIN {X 0,Y 291.546,Z 471.172,A -85,B 0,C 180,E1 -17046.653,E2 -17046.653} C_VEL
LIN {X 0,Y 290.136,Z 466.201,A -85,B 0,C 180,E1 -17049.182,E2 -17049.182} C_VEL
LIN {X 0,Y 288.769,Z 461.464,A -85,B 0,C 180,E1 -17052.072,E2 -17052.072} C_VEL
LIN {X 0,Y 287.454,Z 457.398,A -85,B 0,C 180,E1 -17055.156,E2 -17055.156} C_VEL
LIN {X 0,Y 286.374,Z 454.018,A -85,B 0,C 180,E1 -17058.5,E2 -17058.5} C_VEL
LIN {X 0,Y 285.535,Z 451.627,A -85,B 0,C 180,E1 -17062.023,E2 -17062.023} C_VEL
LIN {X 0,Y 285.207,Z 450.671,A -85,B 0,C 180,E1 -17064.409,E2 -17064.409} C_VEL
LIN {X 0,Y 284.948,Z 450.33,A -85,B 0,C 180,E1 -17068.805,E2 -17068.805} C_VEL
LIN {X 0,Y 285.381,Z 451.035,A -85,B 0,C 180,E1 -17072.101,E2 -17072.101} C_VEL
LIN {X 0,Y 286.139,Z 453.622,A -85,B 0,C 180,E1 -17076.501,E2 -17076.501} C_VEL
LIN {X 0,Y 288.914,Z 457.253,A -85,B 0,C 180,E1 -17077.895,E2 -17077.895} C_VEL
LIN {X 0,Y 290.627,Z 458.905,A -85,B 0,C 180,E1 -17078.639,E2 -17078.639} C_VEL
LIN {X 0,Y 293.486,Z 462.535,A -85,B 0,C 180,E1 -17079.838,E2 -17079.838} C_VEL
LIN {X 0,Y 297.652,Z 468.222,A -85,B 0,C 180,E1 -17081.446,E2 -17081.446} C_VEL
LIN {X 0,Y 302.613,Z 475.657,A -85,B 0,C 180,E1 -17083.164,E2 -17083.164} C_VEL
LIN {X 0,Y 307.344,Z 483.552,A -85,B 0,C 180,E1 -17084.648,E2 -17084.648} C_VEL
LIN {X 0,Y 310.647,Z 490.102,A -85,B 0,C 180,E1 -17085.658,E2 -17085.658} C_VEL
LIN {X 0,Y 305.542,Z 552.833,A -85,B 0,C 180,E1 -17087.884,E2 -17087.884} C_VEL
LIN {X 0,Y 304.219,Z 567.094,A -85,B 0,C 180,E1 -17088.675,E2 -17088.675} C_VEL
LIN {X 0,Y 302.689,Z 579.51,A -85,B 0,C 180,E1 -17089.633,E2 -17089.633} C_VEL
LIN {X 0,Y 300.556,Z 592.042,A -85,B 0,C 180,E1 -17090.891,E2 -17090.891} C_VEL
LIN {X 0,Y 298.299,Z 603.121,A -85,B 0,C 180,E1 -17092.311,E2 -17092.311} C_VEL
LIN {X 0,Y 295.595,Z 614.624,A -85,B 0,C 180,E1 -17094.2,E2 -17094.2} C_VEL
LIN {X 0,Y 293.41,Z 622.857,A -85,B 0,C 180,E1 -17095.879,E2 -17095.879} C_VEL
LIN {X 0,Y 291.148,Z 630.827,A -85,B 0,C 180,E1 -17097.925,E2 -17097.925} C_VEL
LIN {X 0,Y 289.15,Z 637.247,A -85,B 0,C 180,E1 -17100,E2 -17100} C_VEL
LIN {X 0,Y 287.49,Z 642.33,A -85,B 0,C 180,E1 -17102.101,E2 -17102.101} C_VEL
LIN {X 0,Y 286.006,Z 646.43,A -85,B 0,C 180,E1 -17104.333,E2 -17104.333} C_VEL
LIN {X 0,Y 285.313,Z 648.275,A -85,B 0,C 180,E1 -17105.654,E2 -17105.654} C_VEL
LIN {X 0,Y 284.115,Z 650.784,A -85,B 0,C 180,E1 -17108.322,E2 -17108.322} C_VEL
LIN {X 0,Y 283.602,Z 651.592,A -85,B 0,C 180,E1 -17109.989,E2 -17109.989} C_VEL
LIN {X 0,Y 283.25,Z 651.794,A -85,B 0,C 180,E1 -17111.449,E2 -17111.449} C_VEL
LIN {X 0,Y 283.001,Z 651.578,A -85,B 0,C 180,E1 -17112.915,E2 -17112.915} C_VEL
LIN {X 0,Y 282.846,Z 650.918,A -85,B 0,C 180,E1 -17114.387,E2 -17114.387} C_VEL
LIN {X 0,Y 282.712,Z 649.761,A -85,B 0,C 180,E1 -17115.87,E2 -17115.87} C_VEL
LIN {X 0,Y 282.772,Z 647.157,A -85,B 0,C 180,E1 -17118.1,E2 -17118.1} C_VEL
LIN {X 0,Y 282.993,Z 643.396,A -85,B 0,C 180,E1 -17120.346,E2 -17120.346} C_VEL
LIN {X 0,Y 283.399,Z 638.346,A -85,B 0,C 180,E1 -17122.605,E2 -17122.605} C_VEL
LIN {X 0,Y 283.973,Z 631.791,A -85,B 0,C 180,E1 -17124.881,E2 -17124.881} C_VEL
LIN {X 0,Y 284.689,Z 624.56,A -85,B 0,C 180,E1 -17126.884,E2 -17126.884} C_VEL
LIN {X 0,Y 285.672,Z 614.787,A -85,B 0,C 180,E1 -17129.07,E2 -17129.07} C_VEL
LIN {X 0,Y 286.788,Z 604.037,A -85,B 0,C 180,E1 -17130.972,E2 -17130.972} C_VEL
LIN {X 0,Y 287.81,Z 593.387,A -85,B 0,C 180,E1 -17132.494,E2 -17132.494} C_VEL
LIN {X 0,Y 288.76,Z 581.658,A -85,B 0,C 180,E1 -17133.831,E2 -17133.831} C_VEL
LIN {X 0,Y 289.743,Z 568.26,A -85,B 0,C 180,E1 -17135.012,E2 -17135.012} C_VEL
LIN {X 0,Y 290.467,Z 554.774,A -85,B 0,C 180,E1 -17135.873,E2 -17135.873} C_VEL
LIN {X 0,Y 290.95,Z 541.515,A -85,B 0,C 180,E1 -17136.446,E2 -17136.446} C_VEL
LIN {X 0,Y 293.32,Z 473.901,A -85,B 0,C 180,E1 -17138.626,E2 -17138.626} C_VEL
LIN {X 0,Y 284.312,Z 448.07,A -85,B 0,C 180,E1 -17140.071,E2 -17140.071} C_VEL
LIN {X 0,Y 284.236,Z 448.08,A -85,B 0,C 180,E1 -17144.188,E2 -17144.188} C_VEL
LIN {X 0,Y 284.259,Z 448.076,A -85,B 0,C 180,E1 -17148.121,E2 -17148.121} C_VEL
LIN {X 0,Y 284.303,Z 448.072,A -85,B 0,C 180,E1 -17152.283,E2 -17152.283} C_VEL
LIN {X 0,Y 284.309,Z 448.067,A -85,B 0,C 180,E1 -17155.35,E2 -17155.35} C_VEL
LIN {X 0,Y 284.287,Z 448.073,A -85,B 0,C 180,E1 -17158.724,E2 -17158.724} C_VEL
LIN {X 0,Y 284.285,Z 448.071,A -85,B 0,C 180,E1 -17161.984,E2 -17161.984} C_VEL
LIN {X 0,Y 284.326,Z 448.068,A -85,B 0,C 180,E1 -17166.145,E2 -17166.145} C_VEL
LIN {X 0,Y 284.39,Z 448.058,A -85,B 0,C 180,E1 -17169.897,E2 -17169.897} C_VEL
LIN {X 0,Y 284.494,Z 448.049,A -85,B 0,C 180,E1 -17174.459,E2 -17174.459} C_VEL
LIN {X 0,Y 284.484,Z 448.049,A -85,B 0,C 180,E1 -17178.601,E2 -17178.601} C_VEL
LIN {X 0,Y 284.61,Z 448.029,A -85,B 0,C 180,E1 -17181.479,E2 -17181.479} C_VEL
LIN {X 0,Y 284.575,Z 448.038,A -85,B 0,C 180,E1 -17184.33,E2 -17184.33} C_VEL
LIN {X 0,Y 284.852,Z 448.003,A -85,B 0,C 180,E1 -17188.586,E2 -17188.586} C_VEL
LIN {X 0,Y 284.852,Z 448,A -85,B 0,C 180,E1 -17191.413,E2 -17191.413} C_VEL
LIN {X 0,Y 284.675,Z 448.021,A -85,B 0,C 180,E1 -17197.09,E2 -17197.09} C_VEL
LIN {X 0,Y 284.518,Z 448.042,A -85,B 0,C 180,E1 -17199.957,E2 -17199.957} C_VEL
LIN {X 0,Y 284.464,Z 448.051,A -85,B 0,C 180,E1 -17204.303,E2 -17204.303} C_VEL
LIN {X 0,Y 284.375,Z 448.062,A -85,B 0,C 180,E1 -17208.74,E2 -17208.74} C_VEL
LIN {X 0,Y 284.314,Z 448.067,A -85,B 0,C 180,E1 -17211.764,E2 -17211.764} C_VEL
LIN {X 0,Y 284.313,Z 448.068,A -85,B 0,C 180,E1 -17214.848,E2 -17214.848} C_VEL
LIN {X 0,Y 284.288,Z 448.071,A -85,B 0,C 180,E1 -17218.015,E2 -17218.015} C_VEL
LIN {X 0,Y 284.285,Z 448.07,A -85,B 0,C 180,E1 -17221.275,E2 -17221.275} C_VEL
LIN {X 0,Y 284.34,Z 448.063,A -85,B 0,C 180,E1 -17225.347,E2 -17225.347} C_VEL
LIN {X 0,Y 284.3,Z 448.07,A -85,B 0,C 180,E1 -17228.17,E2 -17228.17} C_VEL
LIN {X 0,Y 284.236,Z 448.077,A -85,B 0,C 180,E1 -17232.117,E2 -17232.117} C_VEL
LIN {X 0,Y 284.254,Z 448.076,A -85,B 0,C 180,E1 -17236.189,E2 -17236.189} C_VEL
LIN {X 0,Y 284.305,Z 448.068,A -85,B 0,C 180,E1 -17240.024,E2 -17240.024} C_VEL
LIN {X 0,Y 284.329,Z 448.064,A -85,B 0,C 180,E1 -17243.614,E2 -17243.614} C_VEL
LIN {X 0,Y 284.306,Z 448.068,A -85,B 0,C 180,E1 -17247.189,E2 -17247.189} C_VEL
LIN {X 0,Y 284.354,Z 448.064,A -85,B 0,C 180,E1 -17250.376,E2 -17250.376} C_VEL
LIN {X 0,Y 284.374,Z 448.059,A -85,B 0,C 180,E1 -17253.586,E2 -17253.586} C_VEL
LIN {X 0,Y 284.366,Z 448.064,A -85,B 0,C 180,E1 -17256.707,E2 -17256.707} C_VEL
LIN {X 0,Y 284.403,Z 448.056,A -85,B 0,C 180,E1 -17261.262,E2 -17261.262} C_VEL
LIN {X 0,Y 284.491,Z 448.048,A -85,B 0,C 180,E1 -17264.459,E2 -17264.459} C_VEL
LIN {X 0,Y 284.487,Z 448.049,A -85,B 0,C 180,E1 -17268.602,E2 -17268.602} C_VEL
LIN {X 0,Y 284.654,Z 448.025,A -85,B 0,C 180,E1 -17271.481,E2 -17271.481} C_VEL
LIN {X 0,Y 284.594,Z 448.034,A -85,B 0,C 180,E1 -17274.331,E2 -17274.331} C_VEL
LIN {X 0,Y 284.854,Z 448.004,A -85,B 0,C 180,E1 -17278.586,E2 -17278.586} C_VEL
LIN {X 0,Y 284.829,Z 448.002,A -85,B 0,C 180,E1 -17281.607,E2 -17281.607} C_VEL
LIN {X 0,Y 284.064,Z 448.101,A -85,B 0,C 180,E1 -17282.784,E2 -17282.784} C_VEL
LIN {X 0,Y 281.165,Z 448.462,A -85,B 0,C 180,E1 -17284.703,E2 -17284.703} C_VEL
LIN {X 0,Y 278.752,Z 448.761,A -85,B 0,C 180,E1 -17286.261,E2 -17286.261} C_VEL
LIN {X 0,Y 277.709,Z 448.89,A -85,B 0,C 180,E1 -17287.468,E2 -17287.468} C_VEL
LIN {X 0,Y 277.615,Z 448.901,A -85,B 0,C 180,E1 -17287.877,E2 -17287.877} C_VEL
LIN {X 0,Y 277.506,Z 448.916,A -85,B 0,C 180,E1 -17290.211,E2 -17290.211} C_VEL
LIN {X 0,Y 277.434,Z 448.927,A -85,B 0,C 180,E1 -17294.674,E2 -17294.674} C_VEL
LIN {X 0,Y 277.344,Z 448.936,A -85,B 0,C 180,E1 -17299.234,E2 -17299.234} C_VEL
LIN {X 0,Y 277.292,Z 448.942,A -85,B 0,C 180,E1 -17304.158,E2 -17304.158} C_VEL
LIN {X 0,Y 277.327,Z 448.937,A -85,B 0,C 180,E1 -17307.506,E2 -17307.506} C_VEL
LIN {X 0,Y 277.271,Z 448.947,A -85,B 0,C 180,E1 -17310.482,E2 -17310.482} C_VEL
LIN {X 0,Y 277.247,Z 448.947,A -85,B 0,C 180,E1 -17313.896,E2 -17313.896} C_VEL
LIN {X 0,Y 277.267,Z 448.945,A -85,B 0,C 180,E1 -17317.47,E2 -17317.47} C_VEL
LIN {X 0,Y 277.209,Z 448.952,A -85,B 0,C 180,E1 -17321.237,E2 -17321.237} C_VEL
LIN {X 0,Y 277.216,Z 448.952,A -85,B 0,C 180,E1 -17325.224,E2 -17325.224} C_VEL
LIN {X 0,Y 277.222,Z 448.949,A -85,B 0,C 180,E1 -17329.513,E2 -17329.513} C_VEL
LIN {X 0,Y 277.265,Z 448.948,A -85,B 0,C 180,E1 -17332.531,E2 -17332.531} C_VEL
LIN {X 0,Y 277.295,Z 449.031,A -85,B 0,C 180,E1 -17334.956,E2 -17334.956} C_VEL
LIN {X 0,Y 279.828,Z 461.356,A -85,B 0,C 180,E1 -17338.642,E2 -17338.642} C_VEL
LIN {X 0,Y 282.024,Z 472.134,A -85,B 0,C 180,E1 -17341.74,E2 -17341.74} C_VEL
LIN {X 0,Y 280.74,Z 481.967,A -85,B 0,C 180,E1 -17344.319,E2 -17344.319} C_VEL
LIN {X 0,Y 285.388,Z 530.302,A -85,B 0,C 180,E1 -17346.318,E2 -17346.318} C_VEL
LIN {X 0,Y 283.949,Z 576.292,A -85,B 0,C 180,E1 -17347.872,E2 -17347.872} C_VEL
LIN {X 0,Y 283.22,Z 594.963,A -85,B 0,C 180,E1 -17348.578,E2 -17348.578} C_VEL
LIN {X 0,Y 282.369,Z 607.543,A -85,B 0,C 180,E1 -17349.322,E2 -17349.322} C_VEL
LIN {X 0,Y 281.14,Z 621.393,A -85,B 0,C 180,E1 -17350.467,E2 -17350.467} C_VEL
LIN {X 0,Y 280.068,Z 632.821,A -85,B 0,C 180,E1 -17351.72,E2 -17351.72} C_VEL
LIN {X 0,Y 278.79,Z 645.064,A -85,B 0,C 180,E1 -17353.427,E2 -17353.427} C_VEL
LIN {X 0,Y 277.802,Z 653.963,A -85,B 0,C 180,E1 -17354.971,E2 -17354.971} C_VEL
LIN {X 0,Y 276.998,Z 662.615,A -85,B 0,C 180,E1 -17356.801,E2 -17356.801} C_VEL
LIN {X 0,Y 276.312,Z 671.039,A -85,B 0,C 180,E1 -17359.003,E2 -17359.003} C_VEL
LIN {X 0,Y 275.928,Z 677.78,A -85,B 0,C 180,E1 -17361.21,E2 -17361.21} C_VEL
LIN {X 0,Y 275.804,Z 683.449,A -85,B 0,C 180,E1 -17363.615,E2 -17363.615} C_VEL
LIN {X 0,Y 275.758,Z 687.035,A -85,B 0,C 180,E1 -17365.615,E2 -17365.615} C_VEL
LIN {X 0,Y 275.867,Z 689.04,A -85,B 0,C 180,E1 -17367.08,E2 -17367.08} C_VEL
LIN {X 0,Y 275.95,Z 690.577,A -85,B 0,C 180,E1 -17368.541,E2 -17368.541} C_VEL
LIN {X 0,Y 275.944,Z 691.631,A -85,B 0,C 180,E1 -17370.001,E2 -17370.001} C_VEL
LIN {X 0,Y 275.872,Z 692.197,A -85,B 0,C 180,E1 -17371.46,E2 -17371.46} C_VEL
LIN {X 0,Y 275.582,Z 692.314,A -85,B 0,C 180,E1 -17372.924,E2 -17372.924} C_VEL
LIN {X 0,Y 275.496,Z 692.026,A -85,B 0,C 180,E1 -17374.39,E2 -17374.39} C_VEL
LIN {X 0,Y 275.447,Z 691.293,A -85,B 0,C 180,E1 -17375.858,E2 -17375.858} C_VEL
LIN {X 0,Y 275.688,Z 688.545,A -85,B 0,C 180,E1 -17378.799,E2 -17378.799} C_VEL
LIN {X 0,Y 276.199,Z 685.346,A -85,B 0,C 180,E1 -17381.002,E2 -17381.002} C_VEL
LIN {X 0,Y 277.132,Z 681.096,A -85,B 0,C 180,E1 -17383.194,E2 -17383.194} C_VEL
LIN {X 0,Y 278.776,Z 674.76,A -85,B 0,C 180,E1 -17385.725,E2 -17385.725} C_VEL
LIN {X 0,Y 280.595,Z 667.921,A -85,B 0,C 180,E1 -17387.865,E2 -17387.865} C_VEL
LIN {X 0,Y 282.91,Z 659.479,A -85,B 0,C 180,E1 -17389.973,E2 -17389.973} C_VEL
LIN {X 0,Y 285.801,Z 649.195,A -85,B 0,C 180,E1 -17392.025,E2 -17392.025} C_VEL
LIN {X 0,Y 288.535,Z 638.679,A -85,B 0,C 180,E1 -17393.698,E2 -17393.698} C_VEL
LIN {X 0,Y 291.269,Z 627.125,A -85,B 0,C 180,E1 -17395.168,E2 -17395.168} C_VEL
LIN {X 0,Y 293.73,Z 616.001,A -85,B 0,C 180,E1 -17396.273,E2 -17396.273} C_VEL
LIN {X 0,Y 296.369,Z 601.705,A -85,B 0,C 180,E1 -17397.352,E2 -17397.352} C_VEL
LIN {X 0,Y 298.244,Z 587.996,A -85,B 0,C 180,E1 -17398.119,E2 -17398.119} C_VEL
LIN {X 0,Y 300.43,Z 564.315,A -85,B 0,C 180,E1 -17398.984,E2 -17398.984} C_VEL
LIN {X 0,Y 302.637,Z 535.128,A -85,B 0,C 180,E1 -17400.058,E2 -17400.058} C_VEL
LIN {X 0,Y 301.796,Z 520.347,A -85,B 0,C 180,E1 -17401.013,E2 -17401.013} C_VEL
LIN {X 0,Y 299.865,Z 504.857,A -85,B 0,C 180,E1 -17402.29,E2 -17402.29} C_VEL
LIN {X 0,Y 298.663,Z 497.959,A -85,B 0,C 180,E1 -17402.967,E2 -17402.967} C_VEL
LIN {X 0,Y 295.934,Z 491.86,A -85,B 0,C 180,E1 -17404.014,E2 -17404.014} C_VEL
LIN {X 0,Y 293.589,Z 487.023,A -85,B 0,C 180,E1 -17404.937,E2 -17404.937} C_VEL
LIN {X 0,Y 291.201,Z 482.165,A -85,B 0,C 180,E1 -17405.971,E2 -17405.971} C_VEL
LIN {X 0,Y 287.797,Z 475.932,A -85,B 0,C 180,E1 -17407.509,E2 -17407.509} C_VEL
LIN {X 0,Y 284.231,Z 470.089,A -85,B 0,C 180,E1 -17409.289,E2 -17409.289} C_VEL
LIN {X 0,Y 283.728,Z 468.923,A -85,B 0,C 180,E1 -17409.669,E2 -17409.669} C_VEL
LIN {X 0,Y 282.428,Z 464.268,A -85,B 0,C 180,E1 -17412.689,E2 -17412.689} C_VEL
LIN {X 0,Y 281.246,Z 460.686,A -85,B 0,C 180,E1 -17415.598,E2 -17415.598} C_VEL
LIN {X 0,Y 280.133,Z 457.231,A -85,B 0,C 180,E1 -17419.285,E2 -17419.285} C_VEL
LIN {X 0,Y 279.383,Z 454.771,A -85,B 0,C 180,E1 -17423.609,E2 -17423.609} C_VEL
LIN {X 0,Y 279.028,Z 454.182,A -85,B 0,C 180,E1 -17426.349,E2 -17426.349} C_VEL
LIN {X 0,Y 279.066,Z 454.268,A -85,B 0,C 180,E1 -17429.756,E2 -17429.756} C_VEL
LIN {X 0,Y 279.301,Z 454.712,A -85,B 0,C 180,E1 -17431.728,E2 -17431.728} C_VEL
LIN {X 0,Y 279.513,Z 455.625,A -85,B 0,C 180,E1 -17433.543,E2 -17433.543} C_VEL
LIN {X 0,Y 282.06,Z 458.772,A -85,B 0,C 180,E1 -17435.22,E2 -17435.22} C_VEL
LIN {X 0,Y 283.98,Z 460.482,A -85,B 0,C 180,E1 -17436.244,E2 -17436.244} C_VEL
LIN {X 0,Y 286.972,Z 464.138,A -85,B 0,C 180,E1 -17437.771,E2 -17437.771} C_VEL
LIN {X 0,Y 288.075,Z 465.344,A -85,B 0,C 180,E1 -17438.273,E2 -17438.273} C_VEL
LIN {X 0,Y 291.838,Z 470.408,A -85,B 0,C 180,E1 -17439.918,E2 -17439.918} C_VEL
LIN {X 0,Y 294.582,Z 474.282,A -85,B 0,C 180,E1 -17441.012,E2 -17441.012} C_VEL
LIN {X 0,Y 299.012,Z 481.034,A -85,B 0,C 180,E1 -17442.616,E2 -17442.616} C_VEL
LIN {X 0,Y 303.472,Z 488.813,A -85,B 0,C 180,E1 -17444.117,E2 -17444.117} C_VEL
LIN {X 0,Y 305.53,Z 492.988,A -85,B 0,C 180,E1 -17444.792,E2 -17444.792} C_VEL
LIN {X 0,Y 300.254,Z 554.168,A -85,B 0,C 180,E1 -17447.023,E2 -17447.023} C_VEL
LIN {X 0,Y 298.923,Z 567.488,A -85,B 0,C 180,E1 -17447.784,E2 -17447.784} C_VEL
LIN {X 0,Y 297.257,Z 579.859,A -85,B 0,C 180,E1 -17448.752,E2 -17448.752} C_VEL
LIN {X 0,Y 294.937,Z 592.575,A -85,B 0,C 180,E1 -17450.052,E2 -17450.052} C_VEL
LIN {X 0,Y 292.693,Z 602.904,A -85,B 0,C 180,E1 -17451.369,E2 -17451.369} C_VEL
LIN {X 0,Y 290.204,Z 613.239,A -85,B 0,C 180,E1 -17453.045,E2 -17453.045} C_VEL
LIN {X 0,Y 287.359,Z 623.306,A -85,B 0,C 180,E1 -17455.089,E2 -17455.089} C_VEL
LIN {X 0,Y 284.909,Z 631.286,A -85,B 0,C 180,E1 -17457.172,E2 -17457.172} C_VEL
LIN {X 0,Y 282.782,Z 637.75,A -85,B 0,C 180,E1 -17459.288,E2 -17459.288} C_VEL
LIN {X 0,Y 280.971,Z 642.864,A -85,B 0,C 180,E1 -17461.433,E2 -17461.433} C_VEL
LIN {X 0,Y 279.423,Z 646.801,A -85,B 0,C 180,E1 -17463.605,E2 -17463.605} C_VEL
LIN {X 0,Y 278.171,Z 649.657,A -85,B 0,C 180,E1 -17465.8,E2 -17465.8} C_VEL
LIN {X 0,Y 277.035,Z 651.719,A -85,B 0,C 180,E1 -17468.354,E2 -17468.354} C_VEL
LIN {X 0,Y 276.471,Z 652.356,A -85,B 0,C 180,E1 -17470.25,E2 -17470.25} C_VEL
LIN {X 0,Y 276.108,Z 652.394,A -85,B 0,C 180,E1 -17471.749,E2 -17471.749} C_VEL
LIN {X 0,Y 275.775,Z 651.288,A -85,B 0,C 180,E1 -17474.436,E2 -17474.436} C_VEL
LIN {X 0,Y 275.623,Z 649.736,A -85,B 0,C 180,E1 -17476.289,E2 -17476.289} C_VEL
LIN {X 0,Y 275.718,Z 646.801,A -85,B 0,C 180,E1 -17478.58,E2 -17478.58} C_VEL
LIN {X 0,Y 275.99,Z 642.658,A -85,B 0,C 180,E1 -17480.886,E2 -17480.886} C_VEL
LIN {X 0,Y 276.411,Z 637.369,A -85,B 0,C 180,E1 -17483.131,E2 -17483.131} C_VEL
LIN {X 0,Y 277.1,Z 630.127,A -85,B 0,C 180,E1 -17485.541,E2 -17485.541} C_VEL
LIN {X 0,Y 277.968,Z 621.689,A -85,B 0,C 180,E1 -17487.757,E2 -17487.757} C_VEL
LIN {X 0,Y 278.976,Z 611.823,A -85,B 0,C 180,E1 -17489.838,E2 -17489.838} C_VEL
LIN {X 0,Y 279.979,Z 601.948,A -85,B 0,C 180,E1 -17491.521,E2 -17491.521} C_VEL
LIN {X 0,Y 281.113,Z 590.026,A -85,B 0,C 180,E1 -17493.154,E2 -17493.154} C_VEL
LIN {X 0,Y 282.158,Z 577.323,A -85,B 0,C 180,E1 -17494.517,E2 -17494.517} C_VEL
LIN {X 0,Y 283.072,Z 564.233,A -85,B 0,C 180,E1 -17495.584,E2 -17495.584} C_VEL
LIN {X 0,Y 283.665,Z 550.743,A -85,B 0,C 180,E1 -17496.375,E2 -17496.375} C_VEL
LIN {X 0,Y 284.421,Z 528.119,A -85,B 0,C 180,E1 -17497.201,E2 -17497.201} C_VEL
LIN {X 0,Y 286.41,Z 475.232,A -85,B 0,C 180,E1 -17498.962,E2 -17498.962} C_VEL
LIN {X 0,Y 277.259,Z 448.95,A -85,B 0,C 180,E1 -17500.463,E2 -17500.463} C_VEL
LIN {X 0,Y 277.197,Z 448.955,A -85,B 0,C 180,E1 -17504.772,E2 -17504.772} C_VEL
LIN {X 0,Y 277.196,Z 448.956,A -85,B 0,C 180,E1 -17508.76,E2 -17508.76} C_VEL
LIN {X 0,Y 277.25,Z 448.95,A -85,B 0,C 180,E1 -17512.527,E2 -17512.527} C_VEL
LIN {X 0,Y 277.248,Z 448.949,A -85,B 0,C 180,E1 -17516.104,E2 -17516.104} C_VEL
LIN {X 0,Y 277.264,Z 448.945,A -85,B 0,C 180,E1 -17519.538,E2 -17519.538} C_VEL
LIN {X 0,Y 277.294,Z 448.942,A -85,B 0,C 180,E1 -17522.857,E2 -17522.857} C_VEL
LIN {X 0,Y 277.287,Z 448.944,A -85,B 0,C 180,E1 -17526.075,E2 -17526.075} C_VEL
LIN {X 0,Y 277.347,Z 448.936,A -85,B 0,C 180,E1 -17530.766,E2 -17530.766} C_VEL
LIN {X 0,Y 277.437,Z 448.924,A -85,B 0,C 180,E1 -17535.325,E2 -17535.325} C_VEL
LIN {X 0,Y 277.459,Z 448.92,A -85,B 0,C 180,E1 -17539.786,E2 -17539.786} C_VEL
LIN {X 0,Y 277.603,Z 448.906,A -85,B 0,C 180,E1 -17542.727,E2 -17542.727} C_VEL
LIN {X 0,Y 277.818,Z 448.879,A -85,B 0,C 180,E1 -17548.55,E2 -17548.55} C_VEL
LIN {X 0,Y 277.817,Z 448.876,A -85,B 0,C 180,E1 -17551.449,E2 -17551.449} C_VEL
LIN {X 0,Y 277.629,Z 448.898,A -85,B 0,C 180,E1 -17557.271,E2 -17557.271} C_VEL
LIN {X 0,Y 277.461,Z 448.922,A -85,B 0,C 180,E1 -17560.212,E2 -17560.212} C_VEL
LIN {X 0,Y 277.41,Z 448.929,A -85,B 0,C 180,E1 -17564.675,E2 -17564.675} C_VEL
LIN {X 0,Y 277.324,Z 448.938,A -85,B 0,C 180,E1 -17569.235,E2 -17569.235} C_VEL
LIN {X 0,Y 277.286,Z 448.942,A -85,B 0,C 180,E1 -17573.924,E2 -17573.924} C_VEL
LIN {X 0,Y 277.273,Z 448.943,A -85,B 0,C 180,E1 -17577.484,E2 -17577.484} C_VEL
LIN {X 0,Y 277.247,Z 448.952,A -85,B 0,C 180,E1 -17580.472,E2 -17580.472} C_VEL
LIN {X 0,Y 277.246,Z 448.946,A -85,B 0,C 180,E1 -17583.895,E2 -17583.895} C_VEL
LIN {X 0,Y 277.26,Z 448.946,A -85,B 0,C 180,E1 -17587.47,E2 -17587.47} C_VEL
LIN {X 0,Y 277.183,Z 448.955,A -85,B 0,C 180,E1 -17591.241,E2 -17591.241} C_VEL
LIN {X 0,Y 277.2,Z 448.953,A -85,B 0,C 180,E1 -17595.226,E2 -17595.226} C_VEL
LIN {X 0,Y 277.221,Z 448.95,A -85,B 0,C 180,E1 -17599.512,E2 -17599.512} C_VEL
LIN {X 0,Y 277.264,Z 448.948,A -85,B 0,C 180,E1 -17602.53,E2 -17602.53} C_VEL
LIN {X 0,Y 277.246,Z 448.949,A -85,B 0,C 180,E1 -17606.104,E2 -17606.104} C_VEL
LIN {X 0,Y 277.26,Z 448.944,A -85,B 0,C 180,E1 -17609.538,E2 -17609.538} C_VEL
LIN {X 0,Y 277.355,Z 448.937,A -85,B 0,C 180,E1 -17612.864,E2 -17612.864} C_VEL
LIN {X 0,Y 277.327,Z 448.938,A -85,B 0,C 180,E1 -17616.079,E2 -17616.079} C_VEL
LIN {X 0,Y 277.344,Z 448.939,A -85,B 0,C 180,E1 -17620.766,E2 -17620.766} C_VEL
LIN {X 0,Y 277.434,Z 448.924,A -85,B 0,C 180,E1 -17625.326,E2 -17625.326} C_VEL
LIN {X 0,Y 277.506,Z 448.915,A -85,B 0,C 180,E1 -17629.789,E2 -17629.789} C_VEL
LIN {X 0,Y 277.645,Z 448.902,A -85,B 0,C 180,E1 -17632.729,E2 -17632.729} C_VEL
LIN {X 0,Y 277.82,Z 448.879,A -85,B 0,C 180,E1 -17638.551,E2 -17638.551} C_VEL
LIN {X 0,Y 277.803,Z 448.877,A -85,B 0,C 180,E1 -17641.567,E2 -17641.567} C_VEL
LIN {X 0,Y 277.653,Z 448.897,A -85,B 0,C 180,E1 -17647.271,E2 -17647.271} C_VEL
LIN {X 0,Y 277.615,Z 448.901,A -85,B 0,C 180,E1 -17647.877,E2 -17647.877} C_VEL
LIN {X 0,Y 276.899,Z 448.994,A -85,B 0,C 180,E1 -17649.088,E2 -17649.088} C_VEL
LIN {X 0,Y 273.943,Z 449.36,A -85,B 0,C 180,E1 -17651.056,E2 -17651.056} C_VEL
LIN {X 0,Y 271.466,Z 449.671,A -85,B 0,C 180,E1 -17652.657,E2 -17652.657} C_VEL
LIN {X 0,Y 270.429,Z 449.795,A -85,B 0,C 180,E1 -17653.9,E2 -17653.9} C_VEL
LIN {X 0,Y 270.357,Z 449.802,A -85,B 0,C 180,E1 -17654.321,E2 -17654.321} C_VEL
LIN {X 0,Y 270.29,Z 449.815,A -85,B 0,C 180,E1 -17658.181,E2 -17658.181} C_VEL
LIN {X 0,Y 270.213,Z 449.823,A -85,B 0,C 180,E1 -17661.354,E2 -17661.354} C_VEL
LIN {X 0,Y 270.238,Z 449.823,A -85,B 0,C 180,E1 -17664.589,E2 -17664.589} C_VEL
LIN {X 0,Y 270.272,Z 449.816,A -85,B 0,C 180,E1 -17667.909,E2 -17667.909} C_VEL
LIN {X 0,Y 270.184,Z 449.826,A -85,B 0,C 180,E1 -17671.348,E2 -17671.348} C_VEL
LIN {X 0,Y 270.201,Z 449.828,A -85,B 0,C 180,E1 -17674.906,E2 -17674.906} C_VEL
LIN {X 0,Y 270.197,Z 449.829,A -85,B 0,C 180,E1 -17678.711,E2 -17678.711} C_VEL
LIN {X 0,Y 270.171,Z 449.83,A -85,B 0,C 180,E1 -17683.251,E2 -17683.251} C_VEL
LIN {X 0,Y 270.174,Z 449.827,A -85,B 0,C 180,E1 -17687.443,E2 -17687.443} C_VEL
LIN {X 0,Y 270.207,Z 449.824,A -85,B 0,C 180,E1 -17691.375,E2 -17691.375} C_VEL
LIN {X 0,Y 270.267,Z 449.864,A -85,B 0,C 180,E1 -17694.649,E2 -17694.649} C_VEL
LIN {X 0,Y 272.801,Z 462.275,A -85,B 0,C 180,E1 -17698.462,E2 -17698.462} C_VEL
LIN {X 0,Y 274.876,Z 472.063,A -85,B 0,C 180,E1 -17701.354,E2 -17701.354} C_VEL
LIN {X 0,Y 274.555,Z 476.46,A -85,B 0,C 180,E1 -17702.564,E2 -17702.564} C_VEL
LIN {X 0,Y 273.838,Z 481.35,A -85,B 0,C 180,E1 -17703.891,E2 -17703.891} C_VEL
LIN {X 0,Y 278.17,Z 528.241,A -85,B 0,C 180,E1 -17705.882,E2 -17705.882} C_VEL
LIN {X 0,Y 278.562,Z 533.517,A -85,B 0,C 180,E1 -17706.094,E2 -17706.094} C_VEL
LIN {X 0,Y 276.416,Z 591.678,A -85,B 0,C 180,E1 -17708.171,E2 -17708.171} C_VEL
LIN {X 0,Y 275.524,Z 605.771,A -85,B 0,C 180,E1 -17708.98,E2 -17708.98} C_VEL
LIN {X 0,Y 274.399,Z 617.921,A -85,B 0,C 180,E1 -17709.967,E2 -17709.967} C_VEL
LIN {X 0,Y 273.271,Z 629.95,A -85,B 0,C 180,E1 -17711.248,E2 -17711.248} C_VEL
LIN {X 0,Y 272.162,Z 640.453,A -85,B 0,C 180,E1 -17712.654,E2 -17712.654} C_VEL
LIN {X 0,Y 271.122,Z 649.878,A -85,B 0,C 180,E1 -17714.207,E2 -17714.207} C_VEL
LIN {X 0,Y 270.22,Z 659.163,A -85,B 0,C 180,E1 -17716.08,E2 -17716.08} C_VEL
LIN {X 0,Y 269.395,Z 668.21,A -85,B 0,C 180,E1 -17718.336,E2 -17718.336} C_VEL
LIN {X 0,Y 268.934,Z 675.381,A -85,B 0,C 180,E1 -17720.6,E2 -17720.6} C_VEL
LIN {X 0,Y 268.761,Z 681.431,A -85,B 0,C 180,E1 -17723.035,E2 -17723.035} C_VEL
LIN {X 0,Y 268.706,Z 686.035,A -85,B 0,C 180,E1 -17725.5,E2 -17725.5} C_VEL
LIN {X 0,Y 268.804,Z 688.132,A -85,B 0,C 180,E1 -17727.003,E2 -17727.003} C_VEL
LIN {X 0,Y 268.895,Z 689.734,A -85,B 0,C 180,E1 -17728.503,E2 -17728.503} C_VEL
LIN {X 0,Y 268.89,Z 690.874,A -85,B 0,C 180,E1 -17730.001,E2 -17730.001} C_VEL
LIN {X 0,Y 268.808,Z 691.53,A -85,B 0,C 180,E1 -17731.499,E2 -17731.499} C_VEL
LIN {X 0,Y 268.409,Z 691.476,A -85,B 0,C 180,E1 -17734.506,E2 -17734.506} C_VEL
LIN {X 0,Y 268.353,Z 690.834,A -85,B 0,C 180,E1 -17736.014,E2 -17736.014} C_VEL
LIN {X 0,Y 268.4,Z 689.76,A -85,B 0,C 180,E1 -17737.524,E2 -17737.524} C_VEL
LIN {X 0,Y 268.643,Z 688.245,A -85,B 0,C 180,E1 -17739.031,E2 -17739.031} C_VEL
LIN {X 0,Y 269.433,Z 683.962,A -85,B 0,C 180,E1 -17742.045,E2 -17742.045} C_VEL
LIN {X 0,Y 270.686,Z 679.531,A -85,B 0,C 180,E1 -17744.28,E2 -17744.28} C_VEL
LIN {X 0,Y 272.476,Z 672.88,A -85,B 0,C 180,E1 -17746.869,E2 -17746.869} C_VEL
LIN {X 0,Y 274.993,Z 664.456,A -85,B 0,C 180,E1 -17749.405,E2 -17749.405} C_VEL
LIN {X 0,Y 277.72,Z 655.482,A -85,B 0,C 180,E1 -17751.528,E2 -17751.528} C_VEL
LIN {X 0,Y 280.965,Z 644.425,A -85,B 0,C 180,E1 -17753.593,E2 -17753.593} C_VEL
LIN {X 0,Y 283.978,Z 632.979,A -85,B 0,C 180,E1 -17755.272,E2 -17755.272} C_VEL
LIN {X 0,Y 286.766,Z 621.856,A -85,B 0,C 180,E1 -17756.569,E2 -17756.569} C_VEL
LIN {X 0,Y 289.481,Z 609.728,A -85,B 0,C 180,E1 -17757.667,E2 -17757.667} C_VEL
LIN {X 0,Y 291.895,Z 596.195,A -85,B 0,C 180,E1 -17758.59,E2 -17758.59} C_VEL
LIN {X 0,Y 293.437,Z 584.17,A -85,B 0,C 180,E1 -17759.209,E2 -17759.209} C_VEL
LIN {X 0,Y 297.624,Z 536.156,A -85,B 0,C 180,E1 -17760.999,E2 -17760.999} C_VEL
LIN {X 0,Y 296.892,Z 522.22,A -85,B 0,C 180,E1 -17761.942,E2 -17761.942} C_VEL
LIN {X 0,Y 295.3,Z 507.836,A -85,B 0,C 180,E1 -17763.167,E2 -17763.167} C_VEL
LIN {X 0,Y 294.387,Z 502.047,A -85,B 0,C 180,E1 -17763.759,E2 -17763.759} C_VEL
LIN {X 0,Y 290.822,Z 493.699,A -85,B 0,C 180,E1 -17765.257,E2 -17765.257} C_VEL
LIN {X 0,Y 287.701,Z 487.381,A -85,B 0,C 180,E1 -17766.642,E2 -17766.642} C_VEL
LIN {X 0,Y 284.66,Z 481.516,A -85,B 0,C 180,E1 -17768.148,E2 -17768.148} C_VEL
LIN {X 0,Y 281.4,Z 475.793,A -85,B 0,C 180,E1 -17769.925,E2 -17769.925} C_VEL
LIN {X 0,Y 275.995,Z 466.717,A -85,B 0,C 180,E1 -17773.639,E2 -17773.639} C_VEL
LIN {X 0,Y 274.953,Z 463.67,A -85,B 0,C 180,E1 -17776.359,E2 -17776.359} C_VEL
LIN {X 0,Y 274.434,Z 461.907,A -85,B 0,C 180,E1 -17778.253,E2 -17778.253} C_VEL
LIN {X 0,Y 273.582,Z 459.449,A -85,B 0,C 180,E1 -17781.936,E2 -17781.936} C_VEL
LIN {X 0,Y 273.419,Z 458.579,A -85,B 0,C 180,E1 -17783.758,E2 -17783.758} C_VEL
LIN {X 0,Y 272.992,Z 457.999,A -85,B 0,C 180,E1 -17788.165,E2 -17788.165} C_VEL
LIN {X 0,Y 273.193,Z 458.235,A -85,B 0,C 180,E1 -17789.357,E2 -17789.357} C_VEL
LIN {X 0,Y 277.243,Z 462.052,A -85,B 0,C 180,E1 -17793.055,E2 -17793.055} C_VEL
LIN {X 0,Y 280.284,Z 465.692,A -85,B 0,C 180,E1 -17795.125,E2 -17795.125} C_VEL
LIN {X 0,Y 281.757,Z 467.136,A -85,B 0,C 180,E1 -17795.94,E2 -17795.94} C_VEL
LIN {X 0,Y 284.763,Z 470.777,A -85,B 0,C 180,E1 -17797.535,E2 -17797.535} C_VEL
LIN {X 0,Y 288.72,Z 476.194,A -85,B 0,C 180,E1 -17799.391,E2 -17799.391} C_VEL
LIN {X 0,Y 293.036,Z 482.479,A -85,B 0,C 180,E1 -17801.15,E2 -17801.15} C_VEL
LIN {X 0,Y 298.077,Z 491.011,A -85,B 0,C 180,E1 -17803.013,E2 -17803.013} C_VEL
LIN {X 0,Y 300.544,Z 495.971,A -85,B 0,C 180,E1 -17803.889,E2 -17803.889} C_VEL
LIN {X 0,Y 295.168,Z 553.996,A -85,B 0,C 180,E1 -17806.05,E2 -17806.05} C_VEL
LIN {X 0,Y 293.866,Z 566.78,A -85,B 0,C 180,E1 -17806.78,E2 -17806.78} C_VEL
LIN {X 0,Y 292.189,Z 578.588,A -85,B 0,C 180,E1 -17807.674,E2 -17807.674} C_VEL
LIN {X 0,Y 290.101,Z 590.317,A -85,B 0,C 180,E1 -17808.825,E2 -17808.825} C_VEL
LIN {X 0,Y 287.388,Z 602.239,A -85,B 0,C 180,E1 -17810.321,E2 -17810.321} C_VEL
LIN {X 0,Y 284.735,Z 612.635,A -85,B 0,C 180,E1 -17811.987,E2 -17811.987} C_VEL
LIN {X 0,Y 281.955,Z 622.12,A -85,B 0,C 180,E1 -17813.883,E2 -17813.883} C_VEL
LIN {X 0,Y 279.656,Z 629.346,A -85,B 0,C 180,E1 -17815.676,E2 -17815.676} C_VEL
LIN {X 0,Y 277.219,Z 636.306,A -85,B 0,C 180,E1 -17817.821,E2 -17817.821} C_VEL
LIN {X 0,Y 275.092,Z 641.862,A -85,B 0,C 180,E1 -17820,E2 -17820} C_VEL
LIN {X 0,Y 273.32,Z 646.204,A -85,B 0,C 180,E1 -17822.21,E2 -17822.21} C_VEL
LIN {X 0,Y 271.861,Z 649.426,A -85,B 0,C 180,E1 -17824.448,E2 -17824.448} C_VEL
LIN {X 0,Y 271.025,Z 650.976,A -85,B 0,C 180,E1 -17825.954,E2 -17825.954} C_VEL
LIN {X 0,Y 269.964,Z 652.568,A -85,B 0,C 180,E1 -17828.401,E2 -17828.401} C_VEL
LIN {X 0,Y 269.324,Z 653.042,A -85,B 0,C 180,E1 -17830.525,E2 -17830.525} C_VEL
LIN {X 0,Y 268.958,Z 652.848,A -85,B 0,C 180,E1 -17832.066,E2 -17832.066} C_VEL
LIN {X 0,Y 268.674,Z 651.593,A -85,B 0,C 180,E1 -17834.566,E2 -17834.566} C_VEL
LIN {X 0,Y 268.552,Z 648.58,A -85,B 0,C 180,E1 -17837.515,E2 -17837.515} C_VEL
LIN {X 0,Y 268.756,Z 644.903,A -85,B 0,C 180,E1 -17839.874,E2 -17839.874} C_VEL
LIN {X 0,Y 269.128,Z 639.95,A -85,B 0,C 180,E1 -17842.25,E2 -17842.25} C_VEL
LIN {X 0,Y 269.72,Z 633.548,A -85,B 0,C 180,E1 -17844.639,E2 -17844.639} C_VEL
LIN {X 0,Y 270.524,Z 625.304,A -85,B 0,C 180,E1 -17847.041,E2 -17847.041} C_VEL
LIN {X 0,Y 271.406,Z 616.58,A -85,B 0,C 180,E1 -17849.091,E2 -17849.091} C_VEL
LIN {X 0,Y 272.548,Z 606.26,A -85,B 0,C 180,E1 -17851.046,E2 -17851.046} C_VEL
LIN {X 0,Y 273.659,Z 594.35,A -85,B 0,C 180,E1 -17852.856,E2 -17852.856} C_VEL
LIN {X 0,Y 274.775,Z 582.727,A -85,B 0,C 180,E1 -17854.243,E2 -17854.243} C_VEL
LIN {X 0,Y 275.728,Z 570.229,A -85,B 0,C 180,E1 -17855.414,E2 -17855.414} C_VEL
LIN {X 0,Y 276.522,Z 556.967,A -85,B 0,C 180,E1 -17856.335,E2 -17856.335} C_VEL
LIN {X 0,Y 277.098,Z 542.512,A -85,B 0,C 180,E1 -17857.011,E2 -17857.011} C_VEL
LIN {X 0,Y 279.401,Z 476.317,A -85,B 0,C 180,E1 -17859.309,E2 -17859.309} C_VEL
LIN {X 0,Y 270.187,Z 449.829,A -85,B 0,C 180,E1 -17860.857,E2 -17860.857} C_VEL
LIN {X 0,Y 270.152,Z 449.831,A -85,B 0,C 180,E1 -17865.379,E2 -17865.379} C_VEL
LIN {X 0,Y 270.155,Z 449.831,A -85,B 0,C 180,E1 -17869.43,E2 -17869.43} C_VEL
LIN {X 0,Y 270.22,Z 449.822,A -85,B 0,C 180,E1 -17873.732,E2 -17873.732} C_VEL
LIN {X 0,Y 270.203,Z 449.826,A -85,B 0,C 180,E1 -17876.892,E2 -17876.892} C_VEL
LIN {X 0,Y 270.185,Z 449.831,A -85,B 0,C 180,E1 -17880.381,E2 -17880.381} C_VEL
LIN {X 0,Y 270.205,Z 449.823,A -85,B 0,C 180,E1 -17883.757,E2 -17883.757} C_VEL
LIN {X 0,Y 270.209,Z 449.825,A -85,B 0,C 180,E1 -17887.036,E2 -17887.036} C_VEL
LIN {X 0,Y 270.304,Z 449.815,A -85,B 0,C 180,E1 -17890.244,E2 -17890.244} C_VEL
LIN {X 0,Y 270.405,Z 449.801,A -85,B 0,C 180,E1 -17894.935,E2 -17894.935} C_VEL
LIN {X 0,Y 270.412,Z 449.797,A -85,B 0,C 180,E1 -17899.517,E2 -17899.517} C_VEL
LIN {X 0,Y 270.564,Z 449.784,A -85,B 0,C 180,E1 -17902.537,E2 -17902.537} C_VEL
LIN {X 0,Y 270.784,Z 449.755,A -85,B 0,C 180,E1 -17908.512,E2 -17908.512} C_VEL
LIN {X 0,Y 270.783,Z 449.752,A -85,B 0,C 180,E1 -17911.487,E2 -17911.487} C_VEL
LIN {X 0,Y 270.586,Z 449.775,A -85,B 0,C 180,E1 -17917.461,E2 -17917.461} C_VEL
LIN {X 0,Y 270.413,Z 449.803,A -85,B 0,C 180,E1 -17920.482,E2 -17920.482} C_VEL
LIN {X 0,Y 270.378,Z 449.803,A -85,B 0,C 180,E1 -17925.066,E2 -17925.066} C_VEL
LIN {X 0,Y 270.261,Z 449.818,A -85,B 0,C 180,E1 -17929.758,E2 -17929.758} C_VEL
LIN {X 0,Y 270.226,Z 449.824,A -85,B 0,C 180,E1 -17934.59,E2 -17934.59} C_VEL
LIN {X 0,Y 270.203,Z 449.825,A -85,B 0,C 180,E1 -17937.916,E2 -17937.916} C_VEL
LIN {X 0,Y 270.173,Z 449.828,A -85,B 0,C 180,E1 -17941.349,E2 -17941.349} C_VEL
LIN {X 0,Y 270.2,Z 449.826,A -85,B 0,C 180,E1 -17944.905,E2 -17944.905} C_VEL
LIN {X 0,Y 270.197,Z 449.829,A -85,B 0,C 180,E1 -17948.71,E2 -17948.71} C_VEL
LIN {X 0,Y 270.155,Z 449.83,A -85,B 0,C 180,E1 -17953.247,E2 -17953.247} C_VEL
LIN {X 0,Y 270.17,Z 449.829,A -85,B 0,C 180,E1 -17957.441,E2 -17957.441} C_VEL
LIN {X 0,Y 270.206,Z 449.823,A -85,B 0,C 180,E1 -17961.374,E2 -17961.374} C_VEL
LIN {X 0,Y 270.2,Z 449.826,A -85,B 0,C 180,E1 -17965.094,E2 -17965.094} C_VEL
LIN {X 0,Y 270.199,Z 449.825,A -85,B 0,C 180,E1 -17969.13,E2 -17969.13} C_VEL
LIN {X 0,Y 270.262,Z 449.818,A -85,B 0,C 180,E1 -17972.146,E2 -17972.146} C_VEL
LIN {X 0,Y 270.276,Z 449.815,A -85,B 0,C 180,E1 -17975.519,E2 -17975.519} C_VEL
LIN {X 0,Y 270.301,Z 449.813,A -85,B 0,C 180,E1 -17980.244,E2 -17980.244} C_VEL
LIN {X 0,Y 270.402,Z 449.802,A -85,B 0,C 180,E1 -17984.935,E2 -17984.935} C_VEL
LIN {X 0,Y 270.441,Z 449.794,A -85,B 0,C 180,E1 -17989.519,E2 -17989.519} C_VEL
LIN {X 0,Y 270.604,Z 449.779,A -85,B 0,C 180,E1 -17992.539,E2 -17992.539} C_VEL
LIN {X 0,Y 270.785,Z 449.755,A -85,B 0,C 180,E1 -17998.513,E2 -17998.513} C_VEL
LIN {X 0,Y 270.786,Z 449.752,A -85,B 0,C 180,E1 -18001.487,E2 -18001.487} C_VEL
LIN {X 0,Y 270.611,Z 449.774,A -85,B 0,C 180,E1 -18007.461,E2 -18007.461} C_VEL
LIN {X 0,Y 270.441,Z 449.798,A -85,B 0,C 180,E1 -18010.481,E2 -18010.481} C_VEL
LIN {X 0,Y 270.357,Z 449.802,A -85,B 0,C 180,E1 -18014.321,E2 -18014.321} C_VEL
LIN {X 0,Y 269.73,Z 449.885,A -85,B 0,C 180,E1 -18015.564,E2 -18015.564} C_VEL
LIN {X 0,Y 266.902,Z 450.245,A -85,B 0,C 180,E1 -18017.59,E2 -18017.59} C_VEL
LIN {X 0,Y 264.439,Z 450.552,A -85,B 0,C 180,E1 -18019.236,E2 -18019.236} C_VEL
LIN {X 0,Y 263.324,Z 450.686,A -85,B 0,C 180,E1 -18020.513,E2 -18020.513} C_VEL
LIN {X 0,Y 263.203,Z 450.698,A -85,B 0,C 180,E1 -18020.946,E2 -18020.946} C_VEL
LIN {X 0,Y 263.193,Z 450.699,A -85,B 0,C 180,E1 -18025.293,E2 -18025.293} C_VEL
LIN {X 0,Y 263.18,Z 450.703,A -85,B 0,C 180,E1 -18028.73,E2 -18028.73} C_VEL
LIN {X 0,Y 263.132,Z 450.705,A -85,B 0,C 180,E1 -18032.289,E2 -18032.289} C_VEL
LIN {X 0,Y 263.182,Z 450.703,A -85,B 0,C 180,E1 -18036.764,E2 -18036.764} C_VEL
LIN {X 0,Y 263.125,Z 450.706,A -85,B 0,C 180,E1 -18041.594,E2 -18041.594} C_VEL
LIN {X 0,Y 263.128,Z 450.706,A -85,B 0,C 180,E1 -18046.018,E2 -18046.018} C_VEL
LIN {X 0,Y 263.105,Z 450.708,A -85,B 0,C 180,E1 -18050.128,E2 -18050.128} C_VEL
LIN {X 0,Y 263.256,Z 450.878,A -85,B 0,C 180,E1 -18054.403,E2 -18054.403} C_VEL
LIN {X 0,Y 265.927,Z 464.016,A -85,B 0,C 180,E1 -18058.537,E2 -18058.537} C_VEL
LIN {X 0,Y 267.893,Z 473.486,A -85,B 0,C 180,E1 -18061.395,E2 -18061.395} C_VEL
LIN {X 0,Y 266.976,Z 480.825,A -85,B 0,C 180,E1 -18063.455,E2 -18063.455} C_VEL
LIN {X 0,Y 270.13,Z 518.201,A -85,B 0,C 180,E1 -18065.104,E2 -18065.104} C_VEL
LIN {X 0,Y 271.661,Z 533.371,A -85,B 0,C 180,E1 -18065.761,E2 -18065.761} C_VEL
LIN {X 0,Y 269.46,Z 590.914,A -85,B 0,C 180,E1 -18067.88,E2 -18067.88} C_VEL
LIN {X 0,Y 268.68,Z 603.693,A -85,B 0,C 180,E1 -18068.619,E2 -18068.619} C_VEL
LIN {X 0,Y 267.507,Z 616.284,A -85,B 0,C 180,E1 -18069.629,E2 -18069.629} C_VEL
LIN {X 0,Y 266.308,Z 628.496,A -85,B 0,C 180,E1 -18070.939,E2 -18070.939} C_VEL
LIN {X 0,Y 265.101,Z 640.101,A -85,B 0,C 180,E1 -18072.521,E2 -18072.521} C_VEL
LIN {X 0,Y 264.014,Z 649.757,A -85,B 0,C 180,E1 -18074.166,E2 -18074.166} C_VEL
LIN {X 0,Y 263.127,Z 658.984,A -85,B 0,C 180,E1 -18076.091,E2 -18076.091} C_VEL
LIN {X 0,Y 262.313,Z 667.961,A -85,B 0,C 180,E1 -18078.408,E2 -18078.408} C_VEL
LIN {X 0,Y 261.872,Z 675.07,A -85,B 0,C 180,E1 -18080.734,E2 -18080.734} C_VEL
LIN {X 0,Y 261.709,Z 680.697,A -85,B 0,C 180,E1 -18083.06,E2 -18083.06} C_VEL
LIN {X 0,Y 261.659,Z 684.976,A -85,B 0,C 180,E1 -18085.379,E2 -18085.379} C_VEL
LIN {X 0,Y 261.744,Z 687.193,A -85,B 0,C 180,E1 -18086.922,E2 -18086.922} C_VEL
LIN {X 0,Y 261.841,Z 688.864,A -85,B 0,C 180,E1 -18088.463,E2 -18088.463} C_VEL
LIN {X 0,Y 261.836,Z 690.063,A -85,B 0,C 180,E1 -18090.001,E2 -18090.001} C_VEL
LIN {X 0,Y 261.744,Z 690.814,A -85,B 0,C 180,E1 -18091.539,E2 -18091.539} C_VEL
LIN {X 0,Y 261.416,Z 691.087,A -85,B 0,C 180,E1 -18093.083,E2 -18093.083} C_VEL
LIN {X 0,Y 261.289,Z 690.622,A -85,B 0,C 180,E1 -18095.612,E2 -18095.612} C_VEL
LIN {X 0,Y 261.332,Z 689.367,A -85,B 0,C 180,E1 -18097.728,E2 -18097.728} C_VEL
LIN {X 0,Y 261.58,Z 687.968,A -85,B 0,C 180,E1 -18099.277,E2 -18099.277} C_VEL
LIN {X 0,Y 262.181,Z 685.06,A -85,B 0,C 180,E1 -18101.599,E2 -18101.599} C_VEL
LIN {X 0,Y 263.314,Z 681.134,A -85,B 0,C 180,E1 -18103.9,E2 -18103.9} C_VEL
LIN {X 0,Y 264.845,Z 676.122,A -85,B 0,C 180,E1 -18106.179,E2 -18106.179} C_VEL
LIN {X 0,Y 266.946,Z 669.412,A -85,B 0,C 180,E1 -18108.596,E2 -18108.596} C_VEL
LIN {X 0,Y 269.715,Z 660.908,A -85,B 0,C 180,E1 -18110.996,E2 -18110.996} C_VEL
LIN {X 0,Y 272.84,Z 651.298,A -85,B 0,C 180,E1 -18113.131,E2 -18113.131} C_VEL
LIN {X 0,Y 276.109,Z 640.557,A -85,B 0,C 180,E1 -18115.035,E2 -18115.035} C_VEL
LIN {X 0,Y 279.083,Z 629.868,A -85,B 0,C 180,E1 -18116.551,E2 -18116.551} C_VEL
LIN {X 0,Y 282.098,Z 618.1,A -85,B 0,C 180,E1 -18117.848,E2 -18117.848} C_VEL
LIN {X 0,Y 285.196,Z 604.124,A -85,B 0,C 180,E1 -18119.023,E2 -18119.023} C_VEL
LIN {X 0,Y 287.67,Z 589.15,A -85,B 0,C 180,E1 -18119.955,E2 -18119.955} C_VEL
LIN {X 0,Y 289.404,Z 574.516,A -85,B 0,C 180,E1 -18120.562,E2 -18120.562} C_VEL
LIN {X 0,Y 292.722,Z 537.332,A -85,B 0,C 180,E1 -18121.975,E2 -18121.975} C_VEL
LIN {X 0,Y 292.18,Z 524.105,A -85,B 0,C 180,E1 -18122.908,E2 -18122.908} C_VEL
LIN {X 0,Y 290.793,Z 510.216,A -85,B 0,C 180,E1 -18124.14,E2 -18124.14} C_VEL
LIN {X 0,Y 290.085,Z 505.845,A -85,B 0,C 180,E1 -18124.613,E2 -18124.613} C_VEL
LIN {X 0,Y 286.709,Z 497.746,A -85,B 0,C 180,E1 -18126.176,E2 -18126.176} C_VEL
LIN {X 0,Y 284.267,Z 492.49,A -85,B 0,C 180,E1 -18127.37,E2 -18127.37} C_VEL
LIN {X 0,Y 281.628,Z 487.268,A -85,B 0,C 180,E1 -18128.752,E2 -18128.752} C_VEL
LIN {X 0,Y 278.043,Z 480.649,A -85,B 0,C 180,E1 -18130.903,E2 -18130.903} C_VEL
LIN {X 0,Y 273.535,Z 472.707,A -85,B 0,C 180,E1 -18134.39,E2 -18134.39} C_VEL
LIN {X 0,Y 270.162,Z 467.561,A -85,B 0,C 180,E1 -18138.318,E2 -18138.318} C_VEL
LIN {X 0,Y 269.022,Z 465.139,A -85,B 0,C 180,E1 -18141.382,E2 -18141.382} C_VEL
LIN {X 0,Y 269.012,Z 464.11,A -85,B 0,C 180,E1 -18144.085,E2 -18144.085} C_VEL
LIN {X 0,Y 270.459,Z 464.638,A -85,B 0,C 180,E1 -18147.832,E2 -18147.832} C_VEL
LIN {X 0,Y 271.605,Z 465.209,A -85,B 0,C 180,E1 -18149.266,E2 -18149.266} C_VEL
LIN {X 0,Y 275.565,Z 469.183,A -85,B 0,C 180,E1 -18153.008,E2 -18153.008} C_VEL
LIN {X 0,Y 278.548,Z 472.6,A -85,B 0,C 180,E1 -18155.059,E2 -18155.059} C_VEL
LIN {X 0,Y 282.873,Z 478.055,A -85,B 0,C 180,E1 -18157.472,E2 -18157.472} C_VEL
LIN {X 0,Y 286.218,Z 482.768,A -85,B 0,C 180,E1 -18159.081,E2 -18159.081} C_VEL
LIN {X 0,Y 289.995,Z 488.568,A -85,B 0,C 180,E1 -18160.7,E2 -18160.7} C_VEL
LIN {X 0,Y 294.495,Z 496.502,A -85,B 0,C 180,E1 -18162.472,E2 -18162.472} C_VEL
LIN {X 0,Y 295.721,Z 499.265,A -85,B 0,C 180,E1 -18162.955,E2 -18162.955} C_VEL
LIN {X 0,Y 290.193,Z 555.229,A -85,B 0,C 180,E1 -18165.089,E2 -18165.089} C_VEL
LIN {X 0,Y 288.812,Z 567.797,A -85,B 0,C 180,E1 -18165.826,E2 -18165.826} C_VEL
LIN {X 0,Y 287.002,Z 579.408,A -85,B 0,C 180,E1 -18166.728,E2 -18166.728} C_VEL
LIN {X 0,Y 284.787,Z 590.96,A -85,B 0,C 180,E1 -18167.891,E2 -18167.891} C_VEL
LIN {X 0,Y 281.914,Z 602.885,A -85,B 0,C 180,E1 -18169.405,E2 -18169.405} C_VEL
LIN {X 0,Y 279.336,Z 612.503,A -85,B 0,C 180,E1 -18170.953,E2 -18170.953} C_VEL
LIN {X 0,Y 276.593,Z 621.352,A -85,B 0,C 180,E1 -18172.701,E2 -18172.701} C_VEL
LIN {X 0,Y 274.087,Z 628.646,A -85,B 0,C 180,E1 -18174.482,E2 -18174.482} C_VEL
LIN {X 0,Y 271.387,Z 635.868,A -85,B 0,C 180,E1 -18176.66,E2 -18176.66} C_VEL
LIN {X 0,Y 268.726,Z 642.491,A -85,B 0,C 180,E1 -18179.251,E2 -18179.251} C_VEL
LIN {X 0,Y 266.793,Z 646.806,A -85,B 0,C 180,E1 -18181.509,E2 -18181.509} C_VEL
LIN {X 0,Y 265.199,Z 649.925,A -85,B 0,C 180,E1 -18183.782,E2 -18183.782} C_VEL
LIN {X 0,Y 263.873,Z 652.233,A -85,B 0,C 180,E1 -18186.116,E2 -18186.116} C_VEL
LIN {X 0,Y 262.895,Z 653.431,A -85,B 0,C 180,E1 -18188.453,E2 -18188.453} C_VEL
LIN {X 0,Y 262.165,Z 653.65,A -85,B 0,C 180,E1 -18190.816,E2 -18190.816} C_VEL
LIN {X 0,Y 261.814,Z 653.237,A -85,B 0,C 180,E1 -18192.401,E2 -18192.401} C_VEL
LIN {X 0,Y 261.592,Z 651.851,A -85,B 0,C 180,E1 -18194.716,E2 -18194.716} C_VEL
LIN {X 0,Y 261.495,Z 648.199,A -85,B 0,C 180,E1 -18198.004,E2 -18198.004} C_VEL
LIN {X 0,Y 261.727,Z 644.142,A -85,B 0,C 180,E1 -18200.431,E2 -18200.431} C_VEL
LIN {X 0,Y 262.172,Z 638.736,A -85,B 0,C 180,E1 -18202.874,E2 -18202.874} C_VEL
LIN {X 0,Y 262.821,Z 631.801,A -85,B 0,C 180,E1 -18205.331,E2 -18205.331} C_VEL
LIN {X 0,Y 263.545,Z 624.611,A -85,B 0,C 180,E1 -18207.388,E2 -18207.388} C_VEL
LIN {X 0,Y 264.474,Z 615.814,A -85,B 0,C 180,E1 -18209.446,E2 -18209.446} C_VEL
LIN {X 0,Y 265.688,Z 604.945,A -85,B 0,C 180,E1 -18211.495,E2 -18211.495} C_VEL
LIN {X 0,Y 266.789,Z 593.61,A -85,B 0,C 180,E1 -18213.208,E2 -18213.208} C_VEL
LIN {X 0,Y 267.991,Z 580.324,A -85,B 0,C 180,E1 -18214.777,E2 -18214.777} C_VEL
LIN {X 0,Y 268.977,Z 566.988,A -85,B 0,C 180,E1 -18215.963,E2 -18215.963} C_VEL
LIN {X 0,Y 269.728,Z 553.333,A -85,B 0,C 180,E1 -18216.848,E2 -18216.848} C_VEL
LIN {X 0,Y 270.312,Z 536.35,A -85,B 0,C 180,E1 -18217.544,E2 -18217.544} C_VEL
LIN {X 0,Y 272.534,Z 477.71,A -85,B 0,C 180,E1 -18219.638,E2 -18219.638} C_VEL
LIN {X 0,Y 263.115,Z 450.708,A -85,B 0,C 180,E1 -18221.265,E2 -18221.265} C_VEL
LIN {X 0,Y 263.1,Z 450.712,A -85,B 0,C 180,E1 -18223.989,E2 -18223.989} C_VEL
LIN {X 0,Y 263.117,Z 450.712,A -85,B 0,C 180,E1 -18228.408,E2 -18228.408} C_VEL
LIN {X 0,Y 263.175,Z 450.699,A -85,B 0,C 180,E1 -18233.239,E2 -18233.239} C_VEL
LIN {X 0,Y 263.13,Z 450.706,A -85,B 0,C 180,E1 -18237.711,E2 -18237.711} C_VEL
LIN {X 0,Y 263.15,Z 450.703,A -85,B 0,C 180,E1 -18241.804,E2 -18241.804} C_VEL
LIN {X 0,Y 263.192,Z 450.698,A -85,B 0,C 180,E1 -18245.217,E2 -18245.217} C_VEL
LIN {X 0,Y 263.265,Z 450.689,A -85,B 0,C 180,E1 -18249.693,E2 -18249.693} C_VEL
LIN {X 0,Y 263.353,Z 450.682,A -85,B 0,C 180,E1 -18254.522,E2 -18254.522} C_VEL
LIN {X 0,Y 263.351,Z 450.677,A -85,B 0,C 180,E1 -18259.233,E2 -18259.233} C_VEL
LIN {X 0,Y 263.528,Z 450.659,A -85,B 0,C 180,E1 -18262.337,E2 -18262.337} C_VEL
LIN {X 0,Y 263.748,Z 450.631,A -85,B 0,C 180,E1 -18268.473,E2 -18268.473} C_VEL
LIN {X 0,Y 263.748,Z 450.628,A -85,B 0,C 180,E1 -18271.526,E2 -18271.526} C_VEL
LIN {X 0,Y 263.545,Z 450.652,A -85,B 0,C 180,E1 -18277.662,E2 -18277.662} C_VEL
LIN {X 0,Y 263.355,Z 450.68,A -85,B 0,C 180,E1 -18280.766,E2 -18280.766} C_VEL
LIN {X 0,Y 263.324,Z 450.68,A -85,B 0,C 180,E1 -18285.479,E2 -18285.479} C_VEL
LIN {X 0,Y 263.238,Z 450.695,A -85,B 0,C 180,E1 -18290.308,E2 -18290.308} C_VEL
LIN {X 0,Y 263.17,Z 450.699,A -85,B 0,C 180,E1 -18295.295,E2 -18295.295} C_VEL
LIN {X 0,Y 263.135,Z 450.708,A -85,B 0,C 180,E1 -18298.734,E2 -18298.734} C_VEL
LIN {X 0,Y 263.127,Z 450.708,A -85,B 0,C 180,E1 -18302.288,E2 -18302.288} C_VEL
LIN {X 0,Y 263.179,Z 450.703,A -85,B 0,C 180,E1 -18306.762,E2 -18306.762} C_VEL
LIN {X 0,Y 263.09,Z 450.711,A -85,B 0,C 180,E1 -18309.875,E2 -18309.875} C_VEL
LIN {X 0,Y 263.1,Z 450.709,A -85,B 0,C 180,E1 -18313.988,E2 -18313.988} C_VEL
LIN {X 0,Y 263.123,Z 450.71,A -85,B 0,C 180,E1 -18318.406,E2 -18318.406} C_VEL
LIN {X 0,Y 263.18,Z 450.7,A -85,B 0,C 180,E1 -18323.237,E2 -18323.237} C_VEL
LIN {X 0,Y 263.131,Z 450.705,A -85,B 0,C 180,E1 -18327.712,E2 -18327.712} C_VEL
LIN {X 0,Y 263.195,Z 450.697,A -85,B 0,C 180,E1 -18331.785,E2 -18331.785} C_VEL
LIN {X 0,Y 263.225,Z 450.695,A -85,B 0,C 180,E1 -18335.2,E2 -18335.2} C_VEL
LIN {X 0,Y 263.263,Z 450.688,A -85,B 0,C 180,E1 -18339.693,E2 -18339.693} C_VEL
LIN {X 0,Y 263.35,Z 450.682,A -85,B 0,C 180,E1 -18344.522,E2 -18344.522} C_VEL
LIN {X 0,Y 263.373,Z 450.676,A -85,B 0,C 180,E1 -18349.234,E2 -18349.234} C_VEL
LIN {X 0,Y 263.566,Z 450.654,A -85,B 0,C 180,E1 -18352.338,E2 -18352.338} C_VEL
LIN {X 0,Y 263.75,Z 450.631,A -85,B 0,C 180,E1 -18358.473,E2 -18358.473} C_VEL
LIN {X 0,Y 263.75,Z 450.629,A -85,B 0,C 180,E1 -18361.527,E2 -18361.527} C_VEL
LIN {X 0,Y 263.572,Z 450.65,A -85,B 0,C 180,E1 -18367.662,E2 -18367.662} C_VEL
LIN {X 0,Y 263.374,Z 450.679,A -85,B 0,C 180,E1 -18370.766,E2 -18370.766} C_VEL
LIN {X 0,Y 263.35,Z 450.678,A -85,B 0,C 180,E1 -18375.478,E2 -18375.478} C_VEL
LIN {X 0,Y 263.262,Z 450.691,A -85,B 0,C 180,E1 -18380.307,E2 -18380.307} C_VEL
LIN {X 0,Y 263.203,Z 450.698,A -85,B 0,C 180,E1 -18380.946,E2 -18380.946} C_VEL
LIN {X 0,Y 262.444,Z 450.792,A -85,B 0,C 180,E1 -18382.224,E2 -18382.224} C_VEL
LIN {X 0,Y 259.535,Z 451.154,A -85,B 0,C 180,E1 -18384.307,E2 -18384.307} C_VEL
LIN {X 0,Y 257.154,Z 451.451,A -85,B 0,C 180,E1 -18386.001,E2 -18386.001} C_VEL
LIN {X 0,Y 256.19,Z 451.571,A -85,B 0,C 180,E1 -18387.315,E2 -18387.315} C_VEL
LIN {X 0,Y 256.139,Z 451.576,A -85,B 0,C 180,E1 -18387.759,E2 -18387.759} C_VEL
LIN {X 0,Y 256.082,Z 451.582,A -85,B 0,C 180,E1 -18391.705,E2 -18391.705} C_VEL
LIN {X 0,Y 256.081,Z 451.585,A -85,B 0,C 180,E1 -18395.193,E2 -18395.193} C_VEL
LIN {X 0,Y 256.114,Z 451.58,A -85,B 0,C 180,E1 -18397.271,E2 -18397.271} C_VEL
LIN {X 0,Y 256.055,Z 451.588,A -85,B 0,C 180,E1 -18401.204,E2 -18401.204} C_VEL
LIN {X 0,Y 256.062,Z 451.586,A -85,B 0,C 180,E1 -18405.53,E2 -18405.53} C_VEL
LIN {X 0,Y 256.055,Z 451.589,A -85,B 0,C 180,E1 -18408.797,E2 -18408.797} C_VEL
LIN {X 0,Y 256.13,Z 451.582,A -85,B 0,C 180,E1 -18412.868,E2 -18412.868} C_VEL
LIN {X 0,Y 256.206,Z 451.74,A -85,B 0,C 180,E1 -18414.103,E2 -18414.103} C_VEL
LIN {X 0,Y 258.965,Z 465.396,A -85,B 0,C 180,E1 -18418.515,E2 -18418.515} C_VEL
LIN {X 0,Y 260.855,Z 474.838,A -85,B 0,C 180,E1 -18421.431,E2 -18421.431} C_VEL
LIN {X 0,Y 260.093,Z 480.482,A -85,B 0,C 180,E1 -18423.042,E2 -18423.042} C_VEL
LIN {X 0,Y 262.692,Z 513,A -85,B 0,C 180,E1 -18424.503,E2 -18424.503} C_VEL
LIN {X 0,Y 264.741,Z 533.522,A -85,B 0,C 180,E1 -18425.422,E2 -18425.422} C_VEL
LIN {X 0,Y 262.519,Z 590.155,A -85,B 0,C 180,E1 -18427.574,E2 -18427.574} C_VEL
LIN {X 0,Y 261.72,Z 602.958,A -85,B 0,C 180,E1 -18428.332,E2 -18428.332} C_VEL
LIN {X 0,Y 260.528,Z 615.597,A -85,B 0,C 180,E1 -18429.368,E2 -18429.368} C_VEL
LIN {X 0,Y 259.255,Z 628.623,A -85,B 0,C 180,E1 -18430.811,E2 -18430.811} C_VEL
LIN {X 0,Y 258.008,Z 640.061,A -85,B 0,C 180,E1 -18432.437,E2 -18432.437} C_VEL
LIN {X 0,Y 256.91,Z 649.589,A -85,B 0,C 180,E1 -18434.124,E2 -18434.124} C_VEL
LIN {X 0,Y 256.021,Z 658.733,A -85,B 0,C 180,E1 -18436.102,E2 -18436.102} C_VEL
LIN {X 0,Y 255.243,Z 667.627,A -85,B 0,C 180,E1 -18438.486,E2 -18438.486} C_VEL
LIN {X 0,Y 254.793,Z 674.669,A -85,B 0,C 180,E1 -18440.875,E2 -18440.875} C_VEL
LIN {X 0,Y 254.654,Z 681.065,A -85,B 0,C 180,E1 -18443.663,E2 -18443.663} C_VEL
LIN {X 0,Y 254.638,Z 685.101,A -85,B 0,C 180,E1 -18446.044,E2 -18446.044} C_VEL
LIN {X 0,Y 254.788,Z 687.975,A -85,B 0,C 180,E1 -18448.42,E2 -18448.42} C_VEL
LIN {X 0,Y 254.784,Z 689.248,A -85,B 0,C 180,E1 -18450.001,E2 -18450.001} C_VEL
LIN {X 0,Y 254.679,Z 690.066,A -85,B 0,C 180,E1 -18451.582,E2 -18451.582} C_VEL
LIN {X 0,Y 254.337,Z 690.432,A -85,B 0,C 180,E1 -18453.169,E2 -18453.169} C_VEL
LIN {X 0,Y 254.219,Z 690.157,A -85,B 0,C 180,E1 -18455.591,E2 -18455.591} C_VEL
LIN {X 0,Y 254.283,Z 688.965,A -85,B 0,C 180,E1 -18457.944,E2 -18457.944} C_VEL
LIN {X 0,Y 254.538,Z 687.657,A -85,B 0,C 180,E1 -18459.536,E2 -18459.536} C_VEL
LIN {X 0,Y 255.185,Z 684.876,A -85,B 0,C 180,E1 -18461.921,E2 -18461.921} C_VEL
LIN {X 0,Y 256.391,Z 681.13,A -85,B 0,C 180,E1 -18464.283,E2 -18464.283} C_VEL
LIN {X 0,Y 258.004,Z 676.327,A -85,B 0,C 180,E1 -18466.62,E2 -18466.62} C_VEL
LIN {X 0,Y 260.427,Z 669.351,A -85,B 0,C 180,E1 -18469.264,E2 -18469.264} C_VEL
LIN {X 0,Y 263.157,Z 661.656,A -85,B 0,C 180,E1 -18471.545,E2 -18471.545} C_VEL
LIN {X 0,Y 266.402,Z 652.443,A -85,B 0,C 180,E1 -18473.723,E2 -18473.723} C_VEL
LIN {X 0,Y 269.813,Z 642.125,A -85,B 0,C 180,E1 -18475.661,E2 -18475.661} C_VEL
LIN {X 0,Y 273.256,Z 630.623,A -85,B 0,C 180,E1 -18477.371,E2 -18477.371} C_VEL
LIN {X 0,Y 276.41,Z 619.418,A -85,B 0,C 180,E1 -18478.681,E2 -18478.681} C_VEL
LIN {X 0,Y 279.616,Z 606.116,A -85,B 0,C 180,E1 -18479.867,E2 -18479.867} C_VEL
LIN {X 0,Y 282.201,Z 592.272,A -85,B 0,C 180,E1 -18480.804,E2 -18480.804} C_VEL
LIN {X 0,Y 284.234,Z 577.709,A -85,B 0,C 180,E1 -18481.469,E2 -18481.469} C_VEL
LIN {X 0,Y 288.031,Z 538.681,A -85,B 0,C 180,E1 -18483,E2 -18483} C_VEL
LIN {X 0,Y 287.633,Z 526.113,A -85,B 0,C 180,E1 -18483.91,E2 -18483.91} C_VEL
LIN {X 0,Y 286.481,Z 512.557,A -85,B 0,C 180,E1 -18485.161,E2 -18485.161} C_VEL
LIN {X 0,Y 285.992,Z 509.632,A -85,B 0,C 180,E1 -18485.514,E2 -18485.514} C_VEL
LIN {X 0,Y 283.13,Z 502.674,A -85,B 0,C 180,E1 -18486.922,E2 -18486.922} C_VEL
LIN {X 0,Y 280.975,Z 497.763,A -85,B 0,C 180,E1 -18488.086,E2 -18488.086} C_VEL
LIN {X 0,Y 278.654,Z 492.892,A -85,B 0,C 180,E1 -18489.41,E2 -18489.41} C_VEL
LIN {X 0,Y 275.51,Z 486.796,A -85,B 0,C 180,E1 -18491.432,E2 -18491.432} C_VEL
LIN {X 0,Y 271.551,Z 479.298,A -85,B 0,C 180,E1 -18494.756,E2 -18494.756} C_VEL
LIN {X 0,Y 268.503,Z 474.369,A -85,B 0,C 180,E1 -18498.575,E2 -18498.575} C_VEL
LIN {X 0,Y 267.515,Z 472.045,A -85,B 0,C 180,E1 -18501.527,E2 -18501.527} C_VEL
LIN {X 0,Y 267.475,Z 471.096,A -85,B 0,C 180,E1 -18503.721,E2 -18503.721} C_VEL
LIN {X 0,Y 268.446,Z 471.362,A -85,B 0,C 180,E1 -18506.907,E2 -18506.907} C_VEL
LIN {X 0,Y 269.908,Z 472.024,A -85,B 0,C 180,E1 -18509.052,E2 -18509.052} C_VEL
LIN {X 0,Y 273.515,Z 475.82,A -85,B 0,C 180,E1 -18512.678,E2 -18512.678} C_VEL
LIN {X 0,Y 277.213,Z 480.26,A -85,B 0,C 180,E1 -18515.26,E2 -18515.26} C_VEL
LIN {X 0,Y 280.508,Z 484.654,A -85,B 0,C 180,E1 -18517.157,E2 -18517.157} C_VEL
LIN {X 0,Y 284.666,Z 490.758,A -85,B 0,C 180,E1 -18519.21,E2 -18519.21} C_VEL
LIN {X 0,Y 289.027,Z 498.302,A -85,B 0,C 180,E1 -18521.127,E2 -18521.127} C_VEL
LIN {X 0,Y 291.044,Z 502.228,A -85,B 0,C 180,E1 -18521.962,E2 -18521.962} C_VEL
LIN {X 0,Y 285.375,Z 556.452,A -85,B 0,C 180,E1 -18524.083,E2 -18524.083} C_VEL
LIN {X 0,Y 283.78,Z 569.163,A -85,B 0,C 180,E1 -18524.854,E2 -18524.854} C_VEL
LIN {X 0,Y 281.634,Z 582.213,A -85,B 0,C 180,E1 -18525.918,E2 -18525.918} C_VEL
LIN {X 0,Y 278.914,Z 594.747,A -85,B 0,C 180,E1 -18527.263,E2 -18527.263} C_VEL
LIN {X 0,Y 276.238,Z 604.878,A -85,B 0,C 180,E1 -18528.628,E2 -18528.628} C_VEL
LIN {X 0,Y 273.168,Z 615.113,A -85,B 0,C 180,E1 -18530.373,E2 -18530.373} C_VEL
LIN {X 0,Y 270.348,Z 623.529,A -85,B 0,C 180,E1 -18532.137,E2 -18532.137} C_VEL
LIN {X 0,Y 267.718,Z 630.652,A -85,B 0,C 180,E1 -18533.972,E2 -18533.972} C_VEL
LIN {X 0,Y 264.857,Z 637.596,A -85,B 0,C 180,E1 -18536.196,E2 -18536.196} C_VEL
LIN {X 0,Y 262.411,Z 643.13,A -85,B 0,C 180,E1 -18538.465,E2 -18538.465} C_VEL
LIN {X 0,Y 260.083,Z 647.882,A -85,B 0,C 180,E1 -18541.048,E2 -18541.048} C_VEL
LIN {X 0,Y 258.285,Z 651.111,A -85,B 0,C 180,E1 -18543.564,E2 -18543.564} C_VEL
LIN {X 0,Y 256.703,Z 653.345,A -85,B 0,C 180,E1 -18546.287,E2 -18546.287} C_VEL
LIN {X 0,Y 255.815,Z 654.186,A -85,B 0,C 180,E1 -18548.491,E2 -18548.491} C_VEL
LIN {X 0,Y 254.994,Z 654.123,A -85,B 0,C 180,E1 -18551.124,E2 -18551.124} C_VEL
LIN {X 0,Y 254.692,Z 653.51,A -85,B 0,C 180,E1 -18552.753,E2 -18552.753} C_VEL
LIN {X 0,Y 254.492,Z 652.032,A -85,B 0,C 180,E1 -18554.858,E2 -18554.858} C_VEL
LIN {X 0,Y 254.38,Z 648.875,A -85,B 0,C 180,E1 -18557.692,E2 -18557.692} C_VEL
LIN {X 0,Y 254.594,Z 644.857,A -85,B 0,C 180,E1 -18560.187,E2 -18560.187} C_VEL
LIN {X 0,Y 255.125,Z 638.438,A -85,B 0,C 180,E1 -18563.113,E2 -18563.113} C_VEL
LIN {X 0,Y 255.844,Z 631.026,A -85,B 0,C 180,E1 -18565.715,E2 -18565.715} C_VEL
LIN {X 0,Y 256.762,Z 622.332,A -85,B 0,C 180,E1 -18568.12,E2 -18568.12} C_VEL
LIN {X 0,Y 257.793,Z 612.632,A -85,B 0,C 180,E1 -18570.288,E2 -18570.288} C_VEL
LIN {X 0,Y 258.919,Z 602.042,A -85,B 0,C 180,E1 -18572.188,E2 -18572.188} C_VEL
LIN {X 0,Y 260.094,Z 590.938,A -85,B 0,C 180,E1 -18573.8,E2 -18573.8} C_VEL
LIN {X 0,Y 261.154,Z 578.432,A -85,B 0,C 180,E1 -18575.234,E2 -18575.234} C_VEL
LIN {X 0,Y 262.109,Z 565.74,A -85,B 0,C 180,E1 -18576.35,E2 -18576.35} C_VEL
LIN {X 0,Y 262.795,Z 552.385,A -85,B 0,C 180,E1 -18577.201,E2 -18577.201} C_VEL
LIN {X 0,Y 263.644,Z 529.691,A -85,B 0,C 180,E1 -18578.118,E2 -18578.118} C_VEL
LIN {X 0,Y 265.695,Z 479.22,A -85,B 0,C 180,E1 -18579.979,E2 -18579.979} C_VEL
LIN {X 0,Y 256.087,Z 451.584,A -85,B 0,C 180,E1 -18581.706,E2 -18581.706} C_VEL
LIN {X 0,Y 256.041,Z 451.589,A -85,B 0,C 180,E1 -18585.534,E2 -18585.534} C_VEL
LIN {X 0,Y 256.045,Z 451.59,A -85,B 0,C 180,E1 -18588.794,E2 -18588.794} C_VEL
LIN {X 0,Y 256.1,Z 451.581,A -85,B 0,C 180,E1 -18592.861,E2 -18592.861} C_VEL
LIN {X 0,Y 256.068,Z 451.588,A -85,B 0,C 180,E1 -18596.706,E2 -18596.706} C_VEL
LIN {X 0,Y 256.057,Z 451.591,A -85,B 0,C 180,E1 -18600.392,E2 -18600.392} C_VEL
LIN {X 0,Y 256.135,Z 451.578,A -85,B 0,C 180,E1 -18604.887,E2 -18604.887} C_VEL
LIN {X 0,Y 256.166,Z 451.573,A -85,B 0,C 180,E1 -18609.104,E2 -18609.104} C_VEL
LIN {X 0,Y 256.302,Z 451.557,A -85,B 0,C 180,E1 -18614.085,E2 -18614.085} C_VEL
LIN {X 0,Y 256.293,Z 451.557,A -85,B 0,C 180,E1 -18618.933,E2 -18618.933} C_VEL
LIN {X 0,Y 256.47,Z 451.536,A -85,B 0,C 180,E1 -18622.124,E2 -18622.124} C_VEL
LIN {X 0,Y 256.491,Z 451.534,A -85,B 0,C 180,E1 -18626.858,E2 -18626.858} C_VEL
LIN {X 0,Y 256.745,Z 451.5,A -85,B 0,C 180,E1 -18629.999,E2 -18629.999} C_VEL
LIN {X 0,Y 256.486,Z 451.534,A -85,B 0,C 180,E1 -18633.141,E2 -18633.141} C_VEL
LIN {X 0,Y 256.505,Z 451.53,A -85,B 0,C 180,E1 -18637.873,E2 -18637.873} C_VEL
LIN {X 0,Y 256.29,Z 451.561,A -85,B 0,C 180,E1 -18642.672,E2 -18642.672} C_VEL
LIN {X 0,Y 256.243,Z 451.565,A -85,B 0,C 180,E1 -18646.271,E2 -18646.271} C_VEL
LIN {X 0,Y 256.142,Z 451.577,A -85,B 0,C 180,E1 -18651.11,E2 -18651.11} C_VEL
LIN {X 0,Y 256.134,Z 451.576,A -85,B 0,C 180,E1 -18655.112,E2 -18655.112} C_VEL
LIN {X 0,Y 256.056,Z 451.587,A -85,B 0,C 180,E1 -18659.606,E2 -18659.606} C_VEL
LIN {X 0,Y 256.065,Z 451.584,A -85,B 0,C 180,E1 -18663.293,E2 -18663.293} C_VEL
LIN {X 0,Y 256.111,Z 451.58,A -85,B 0,C 180,E1 -18667.27,E2 -18667.27} C_VEL
LIN {X 0,Y 256.058,Z 451.587,A -85,B 0,C 180,E1 -18672.178,E2 -18672.178} C_VEL
LIN {X 0,Y 256.048,Z 451.592,A -85,B 0,C 180,E1 -18676.67,E2 -18676.67} C_VEL
LIN {X 0,Y 256.07,Z 451.585,A -85,B 0,C 180,E1 -18680.858,E2 -18680.858} C_VEL
LIN {X 0,Y 256.129,Z 451.58,A -85,B 0,C 180,E1 -18682.867,E2 -18682.867} C_VEL
LIN {X 0,Y 256.066,Z 451.589,A -85,B 0,C 180,E1 -18686.707,E2 -18686.707} C_VEL
LIN {X 0,Y 256.102,Z 451.582,A -85,B 0,C 180,E1 -18690.399,E2 -18690.399} C_VEL
LIN {X 0,Y 256.187,Z 451.573,A -85,B 0,C 180,E1 -18694.862,E2 -18694.862} C_VEL
LIN {X 0,Y 256.166,Z 451.573,A -85,B 0,C 180,E1 -18699.105,E2 -18699.105} C_VEL
LIN {X 0,Y 256.299,Z 451.558,A -85,B 0,C 180,E1 -18704.085,E2 -18704.085} C_VEL
LIN {X 0,Y 256.309,Z 451.557,A -85,B 0,C 180,E1 -18708.934,E2 -18708.934} C_VEL
LIN {X 0,Y 256.535,Z 451.529,A -85,B 0,C 180,E1 -18712.127,E2 -18712.127} C_VEL
LIN {X 0,Y 256.713,Z 451.507,A -85,B 0,C 180,E1 -18718.431,E2 -18718.431} C_VEL
LIN {X 0,Y 256.713,Z 451.505,A -85,B 0,C 180,E1 -18721.569,E2 -18721.569} C_VEL
LIN {X 0,Y 256.54,Z 451.527,A -85,B 0,C 180,E1 -18727.873,E2 -18727.873} C_VEL
LIN {X 0,Y 256.309,Z 451.557,A -85,B 0,C 180,E1 -18731.066,E2 -18731.066} C_VEL
LIN {X 0,Y 256.299,Z 451.556,A -85,B 0,C 180,E1 -18735.915,E2 -18735.915} C_VEL
LIN {X 0,Y 256.16,Z 451.575,A -85,B 0,C 180,E1 -18740.93,E2 -18740.93} C_VEL
LIN {X 0,Y 256.171,Z 451.574,A -85,B 0,C 180,E1 -18745.131,E2 -18745.131} C_VEL
LIN {X 0,Y 256.139,Z 451.576,A -85,B 0,C 180,E1 -18747.759,E2 -18747.759} C_VEL
LIN {X 0,Y 255.872,Z 451.615,A -85,B 0,C 180,E1 -18748.637,E2 -18748.637} C_VEL
LIN {X 0,Y 254.551,Z 451.783,A -85,B 0,C 180,E1 -18749.933,E2 -18749.933} C_VEL
LIN {X 0,Y 250.181,Z 452.322,A -85,B 0,C 180,E1 -18752.951,E2 -18752.951} C_VEL
LIN {X 0,Y 249.121,Z 452.452,A -85,B 0,C 180,E1 -18754.303,E2 -18754.303} C_VEL
LIN {X 0,Y 249.039,Z 452.462,A -85,B 0,C 180,E1 -18754.761,E2 -18754.761} C_VEL
LIN {X 0,Y 249.025,Z 452.464,A -85,B 0,C 180,E1 -18758.381,E2 -18758.381} C_VEL
LIN {X 0,Y 249.011,Z 452.469,A -85,B 0,C 180,E1 -18762.794,E2 -18762.794} C_VEL
LIN {X 0,Y 249.018,Z 452.463,A -85,B 0,C 180,E1 -18767.364,E2 -18767.364} C_VEL
LIN {X 0,Y 249.044,Z 452.461,A -85,B 0,C 180,E1 -18772.201,E2 -18772.201} C_VEL
LIN {X 0,Y 249.125,Z 452.561,A -85,B 0,C 180,E1 -18773.792,E2 -18773.792} C_VEL
LIN {X 0,Y 251.968,Z 466.495,A -85,B 0,C 180,E1 -18778.415,E2 -18778.415} C_VEL
LIN {X 0,Y 253.686,Z 474.618,A -85,B 0,C 180,E1 -18781,E2 -18781} C_VEL
LIN {X 0,Y 253.551,Z 477.562,A -85,B 0,C 180,E1 -18781.888,E2 -18781.888} C_VEL
LIN {X 0,Y 253.179,Z 479.919,A -85,B 0,C 180,E1 -18782.584,E2 -18782.584} C_VEL
LIN {X 0,Y 255.797,Z 513.701,A -85,B 0,C 180,E1 -18784.148,E2 -18784.148} C_VEL
LIN {X 0,Y 257.785,Z 535.125,A -85,B 0,C 180,E1 -18785.13,E2 -18785.13} C_VEL
LIN {X 0,Y 255.552,Z 589.916,A -85,B 0,C 180,E1 -18787.302,E2 -18787.302} C_VEL
LIN {X 0,Y 254.667,Z 603.213,A -85,B 0,C 180,E1 -18788.127,E2 -18788.127} C_VEL
LIN {X 0,Y 253.565,Z 614.572,A -85,B 0,C 180,E1 -18789.094,E2 -18789.094} C_VEL
LIN {X 0,Y 252.319,Z 626.877,A -85,B 0,C 180,E1 -18790.474,E2 -18790.474} C_VEL
LIN {X 0,Y 251.147,Z 638.091,A -85,B 0,C 180,E1 -18792.073,E2 -18792.073} C_VEL
LIN {X 0,Y 249.961,Z 648.288,A -85,B 0,C 180,E1 -18793.881,E2 -18793.881} C_VEL
LIN {X 0,Y 248.946,Z 658.385,A -85,B 0,C 180,E1 -18796.116,E2 -18796.116} C_VEL
LIN {X 0,Y 248.242,Z 665.881,A -85,B 0,C 180,E1 -18798.156,E2 -18798.156} C_VEL
LIN {X 0,Y 247.762,Z 673.203,A -85,B 0,C 180,E1 -18800.613,E2 -18800.613} C_VEL
LIN {X 0,Y 247.623,Z 679.624,A -85,B 0,C 180,E1 -18803.399,E2 -18803.399} C_VEL
LIN {X 0,Y 247.61,Z 684.005,A -85,B 0,C 180,E1 -18805.932,E2 -18805.932} C_VEL
LIN {X 0,Y 247.737,Z 687.029,A -85,B 0,C 180,E1 -18808.375,E2 -18808.375} C_VEL
LIN {X 0,Y 247.732,Z 688.423,A -85,B 0,C 180,E1 -18810.001,E2 -18810.001} C_VEL
LIN {X 0,Y 247.615,Z 689.304,A -85,B 0,C 180,E1 -18811.627,E2 -18811.627} C_VEL
LIN {X 0,Y 247.173,Z 689.772,A -85,B 0,C 180,E1 -18814.894,E2 -18814.894} C_VEL
LIN {X 0,Y 247.102,Z 689.387,A -85,B 0,C 180,E1 -18816.533,E2 -18816.533} C_VEL
LIN {X 0,Y 247.514,Z 687.331,A -85,B 0,C 180,E1 -18819.81,E2 -18819.81} C_VEL
LIN {X 0,Y 248.184,Z 684.732,A -85,B 0,C 180,E1 -18822.263,E2 -18822.263} C_VEL
LIN {X 0,Y 249.489,Z 681.162,A -85,B 0,C 180,E1 -18824.687,E2 -18824.687} C_VEL
LIN {X 0,Y 251.173,Z 676.531,A -85,B 0,C 180,E1 -18827.086,E2 -18827.086} C_VEL
LIN {X 0,Y 253.782,Z 669.72,A -85,B 0,C 180,E1 -18829.831,E2 -18829.831} C_VEL
LIN {X 0,Y 256.626,Z 662.454,A -85,B 0,C 180,E1 -18832.121,E2 -18832.121} C_VEL
LIN {X 0,Y 259.369,Z 655.165,A -85,B 0,C 180,E1 -18833.983,E2 -18833.983} C_VEL
LIN {X 0,Y 262.55,Z 646.596,A -85,B 0,C 180,E1 -18835.785,E2 -18835.785} C_VEL
LIN {X 0,Y 266.014,Z 636.339,A -85,B 0,C 180,E1 -18837.539,E2 -18837.539} C_VEL
LIN {X 0,Y 269.506,Z 625.073,A -85,B 0,C 180,E1 -18839.058,E2 -18839.058} C_VEL
LIN {X 0,Y 273.003,Z 612.623,A -85,B 0,C 180,E1 -18840.346,E2 -18840.346} C_VEL
LIN {X 0,Y 276.178,Z 598.809,A -85,B 0,C 180,E1 -18841.445,E2 -18841.445} C_VEL
LIN {X 0,Y 278.474,Z 585.755,A -85,B 0,C 180,E1 -18842.219,E2 -18842.219} C_VEL
LIN {X 0,Y 280.962,Z 564.759,A -85,B 0,C 180,E1 -18843.068,E2 -18843.068} C_VEL
LIN {X 0,Y 283.484,Z 539.873,A -85,B 0,C 180,E1 -18844.068,E2 -18844.068} C_VEL
LIN {X 0,Y 283.267,Z 527.922,A -85,B 0,C 180,E1 -18844.979,E2 -18844.979} C_VEL
